LIN {X 0,Y 624.676,Z 1239.512,A -85,B 0,C 180,E1 23145.411,E2 23145.411} C_VEL
LIN {X 0,Y 624.339,Z 1247.75,A -85,B 0,C 180,E1 23143.336,E2 23143.336} C_VEL
LIN {X 0,Y 624.101,Z 1256.133,A -85,B 0,C 180,E1 23140.806,E2 23140.806} C_VEL
LIN {X 0,Y 623.992,Z 1262.422,A -85,B 0,C 180,E1 23138.387,E2 23138.387} C_VEL
LIN {X 0,Y 623.935,Z 1266.954,A -85,B 0,C 180,E1 23136.074,E2 23136.074} C_VEL
LIN {X 0,Y 623.913,Z 1270.232,A -85,B 0,C 180,E1 23133.586,E2 23133.586} C_VEL
LIN {X 0,Y 623.894,Z 1271.702,A -85,B 0,C 180,E1 23131.196,E2 23131.196} C_VEL
LIN {X 0,Y 623.863,Z 1271.839,A -85,B 0,C 180,E1 23129.268,E2 23129.268} C_VEL
LIN {X 0,Y 623.906,Z 1270.982,A -85,B 0,C 180,E1 23127.339,E2 23127.339} C_VEL
LIN {X 0,Y 623.915,Z 1268.958,A -85,B 0,C 180,E1 23125.223,E2 23125.223} C_VEL
LIN {X 0,Y 623.954,Z 1265.168,A -85,B 0,C 180,E1 23122.823,E2 23122.823} C_VEL
LIN {X 0,Y 623.989,Z 1259.714,A -85,B 0,C 180,E1 23120.41,E2 23120.41} C_VEL
LIN {X 0,Y 624.177,Z 1253.512,A -85,B 0,C 180,E1 23118.265,E2 23118.265} C_VEL
LIN {X 0,Y 624.358,Z 1246.696,A -85,B 0,C 180,E1 23116.293,E2 23116.293} C_VEL
LIN {X 0,Y 624.688,Z 1239.108,A -85,B 0,C 180,E1 23114.404,E2 23114.404} C_VEL
LIN {X 0,Y 625.192,Z 1229.451,A -85,B 0,C 180,E1 23112.313,E2 23112.313} C_VEL
LIN {X 0,Y 626.017,Z 1216.16,A -85,B 0,C 180,E1 23109.822,E2 23109.822} C_VEL
LIN {X 0,Y 626.971,Z 1202.854,A -85,B 0,C 180,E1 23107.666,E2 23107.666} C_VEL
LIN {X 0,Y 628.106,Z 1188.914,A -85,B 0,C 180,E1 23105.654,E2 23105.654} C_VEL
LIN {X 0,Y 629.747,Z 1170.474,A -85,B 0,C 180,E1 23103.303,E2 23103.303} C_VEL
LIN {X 0,Y 631.348,Z 1153.818,A -85,B 0,C 180,E1 23101.431,E2 23101.431} C_VEL
LIN {X 0,Y 633.023,Z 1137.229,A -85,B 0,C 180,E1 23099.748,E2 23099.748} C_VEL
LIN {X 0,Y 635.235,Z 1116.148,A -85,B 0,C 180,E1 23097.835,E2 23097.835} C_VEL
LIN {X 0,Y 637.354,Z 1095.911,A -85,B 0,C 180,E1 23096.221,E2 23096.221} C_VEL
LIN {X 0,Y 639.262,Z 1077.648,A -85,B 0,C 180,E1 23094.913,E2 23094.913} C_VEL
LIN {X 0,Y 641.245,Z 1058.295,A -85,B 0,C 180,E1 23093.668,E2 23093.668} C_VEL
LIN {X 0,Y 643.679,Z 1033.574,A -85,B 0,C 180,E1 23092.268,E2 23092.268} C_VEL
LIN {X 0,Y 645.795,Z 1009.706,A -85,B 0,C 180,E1 23091.115,E2 23091.115} C_VEL
LIN {X 0,Y 647.498,Z 989.405,A -85,B 0,C 180,E1 23090.265,E2 23090.265} C_VEL
LIN {X 0,Y 649.072,Z 968.685,A -85,B 0,C 180,E1 23089.516,E2 23089.516} C_VEL
LIN {X 0,Y 650.69,Z 944.811,A -85,B 0,C 180,E1 23088.789,E2 23088.789} C_VEL
LIN {X 0,Y 652.223,Z 916.346,A -85,B 0,C 180,E1 23088.117,E2 23088.117} C_VEL
LIN {X 0,Y 653.175,Z 892.642,A -85,B 0,C 180,E1 23087.705,E2 23087.705} C_VEL
LIN {X 0,Y 657.264,Z 681.046,A -85,B 0,C 180,E1 23084.878,E2 23084.878} C_VEL
LIN {X 0,Y 661.362,Z 477.486,A -85,B 0,C 180,E1 23082.097,E2 23082.097} C_VEL
LIN {X 0,Y 661.477,Z 466.858,A -85,B 0,C 180,E1 23081.939,E2 23081.939} C_VEL
LIN {X 0,Y 648.53,Z 447.721,A -85,B 0,C 180,E1 23080.328,E2 23080.328} C_VEL
LIN {X 0,Y 637.826,Z 432.872,A -85,B 0,C 180,E1 23078.92,E2 23078.92} C_VEL
LIN {X 0,Y 630.127,Z 422.628,A -85,B 0,C 180,E1 23077.858,E2 23077.858} C_VEL
LIN {X 0,Y 627.185,Z 418.313,A -85,B 0,C 180,E1 23077.403,E2 23077.403} C_VEL
LIN {X 0,Y 625.308,Z 415.032,A -85,B 0,C 180,E1 23076.844,E2 23076.844} C_VEL
LIN {X 0,Y 624.947,Z 413.383,A -85,B 0,C 180,E1 23076.607,E2 23076.607} C_VEL
LIN {X 0,Y 624.889,Z 413.367,A -85,B 0,C 180,E1 23073.507,E2 23073.507} C_VEL
LIN {X 0,Y 624.909,Z 413.359,A -85,B 0,C 180,E1 23070.692,E2 23070.692} C_VEL
LIN {X 0,Y 624.895,Z 413.387,A -85,B 0,C 180,E1 23067.441,E2 23067.441} C_VEL
LIN {X 0,Y 624.897,Z 413.361,A -85,B 0,C 180,E1 23064.584,E2 23064.584} C_VEL
LIN {X 0,Y 624.897,Z 413.369,A -85,B 0,C 180,E1 23061.298,E2 23061.298} C_VEL
LIN {X 0,Y 624.89,Z 413.381,A -85,B 0,C 180,E1 23058.471,E2 23058.471} C_VEL
LIN {X 0,Y 624.908,Z 413.351,A -85,B 0,C 180,E1 23055.26,E2 23055.26} C_VEL
LIN {X 0,Y 624.879,Z 413.387,A -85,B 0,C 180,E1 23052.475,E2 23052.475} C_VEL
LIN {X 0,Y 624.948,Z 413.347,A -85,B 0,C 180,E1 23049.392,E2 23049.392} C_VEL
LIN {X 0,Y 624.875,Z 413.388,A -85,B 0,C 180,E1 23046.431,E2 23046.431} C_VEL
LIN {X 0,Y 624.915,Z 413.355,A -85,B 0,C 180,E1 23043.578,E2 23043.578} C_VEL
LIN {X 0,Y 624.883,Z 413.388,A -85,B 0,C 180,E1 23040.458,E2 23040.458} C_VEL
LIN {X 0,Y 624.875,Z 413.369,A -85,B 0,C 180,E1 23037.799,E2 23037.799} C_VEL
LIN {X 0,Y 624.922,Z 413.381,A -85,B 0,C 180,E1 23034.675,E2 23034.675} C_VEL
LIN {X 0,Y 624.866,Z 413.376,A -85,B 0,C 180,E1 23031.905,E2 23031.905} C_VEL
LIN {X 0,Y 624.916,Z 413.371,A -85,B 0,C 180,E1 23029.024,E2 23029.024} C_VEL
LIN {X 0,Y 624.871,Z 413.371,A -85,B 0,C 180,E1 23025.923,E2 23025.923} C_VEL
LIN {X 0,Y 624.871,Z 413.378,A -85,B 0,C 180,E1 23023.26,E2 23023.26} C_VEL
LIN {X 0,Y 624.915,Z 413.353,A -85,B 0,C 180,E1 23020.171,E2 23020.171} C_VEL
LIN {X 0,Y 624.862,Z 413.39,A -85,B 0,C 180,E1 23017.316,E2 23017.316} C_VEL
LIN {X 0,Y 624.923,Z 413.354,A -85,B 0,C 180,E1 23014.405,E2 23014.405} C_VEL
LIN {X 0,Y 624.867,Z 413.387,A -85,B 0,C 180,E1 23011.416,E2 23011.416} C_VEL
LIN {X 0,Y 624.859,Z 413.377,A -85,B 0,C 180,E1 23008.872,E2 23008.872} C_VEL
LIN {X 0,Y 624.933,Z 413.356,A -85,B 0,C 180,E1 23005.833,E2 23005.833} C_VEL
LIN {X 0,Y 624.919,Z 413.433,A -85,B 0,C 180,E1 23004.111,E2 23004.111} C_VEL
LIN {X 0,Y 626.366,Z 417.088,A -85,B 0,C 180,E1 23003.57,E2 23003.57} C_VEL
LIN {X 0,Y 627.307,Z 418.786,A -85,B 0,C 180,E1 23003.29,E2 23003.29} C_VEL
LIN {X 0,Y 631.778,Z 427.462,A -85,B 0,C 180,E1 23001.971,E2 23001.971} C_VEL
LIN {X 0,Y 645.743,Z 446.959,A -85,B 0,C 180,E1 23000.086,E2 23000.086} C_VEL
LIN {X 0,Y 661.259,Z 469.603,A -85,B 0,C 180,E1 22998.147,E2 22998.147} C_VEL
LIN {X 0,Y 661.67,Z 470.762,A -85,B 0,C 180,E1 22998.089,E2 22998.089} C_VEL
LIN {X 0,Y 657.702,Z 668.474,A -85,B 0,C 180,E1 22995.381,E2 22995.381} C_VEL
LIN {X 0,Y 653.463,Z 894.03,A -85,B 0,C 180,E1 22992.376,E2 22992.376} C_VEL
LIN {X 0,Y 652.5,Z 920.141,A -85,B 0,C 180,E1 22991.957,E2 22991.957} C_VEL
LIN {X 0,Y 651.364,Z 942.815,A -85,B 0,C 180,E1 22991.471,E2 22991.471} C_VEL
LIN {X 0,Y 649.955,Z 966.319,A -85,B 0,C 180,E1 22990.835,E2 22990.835} C_VEL
LIN {X 0,Y 647.891,Z 994.546,A -85,B 0,C 180,E1 22989.879,E2 22989.879} C_VEL
LIN {X 0,Y 646.07,Z 1016.552,A -85,B 0,C 180,E1 22988.98,E2 22988.98} C_VEL
LIN {X 0,Y 644.268,Z 1036.777,A -85,B 0,C 180,E1 22988.029,E2 22988.029} C_VEL
LIN {X 0,Y 642.215,Z 1058.311,A -85,B 0,C 180,E1 22986.879,E2 22986.879} C_VEL
LIN {X 0,Y 639.686,Z 1083.572,A -85,B 0,C 180,E1 22985.32,E2 22985.32} C_VEL
LIN {X 0,Y 637.629,Z 1103.286,A -85,B 0,C 180,E1 22983.93,E2 22983.93} C_VEL
LIN {X 0,Y 635.755,Z 1121.099,A -85,B 0,C 180,E1 22982.535,E2 22982.535} C_VEL
LIN {X 0,Y 633.772,Z 1140.151,A -85,B 0,C 180,E1 22980.878,E2 22980.878} C_VEL
LIN {X 0,Y 631.607,Z 1161.096,A -85,B 0,C 180,E1 22978.815,E2 22978.815} C_VEL
LIN {X 0,Y 630.115,Z 1176.719,A -85,B 0,C 180,E1 22977.088,E2 22977.088} C_VEL
LIN {X 0,Y 628.633,Z 1192.732,A -85,B 0,C 180,E1 22975.126,E2 22975.126} C_VEL
LIN {X 0,Y 627.231,Z 1209.562,A -85,B 0,C 180,E1 22972.787,E2 22972.787} C_VEL
LIN {X 0,Y 626.247,Z 1222.456,A -85,B 0,C 180,E1 22970.756,E2 22970.756} C_VEL
LIN {X 0,Y 625.503,Z 1233.839,A -85,B 0,C 180,E1 22968.738,E2 22968.738} C_VEL
LIN {X 0,Y 624.848,Z 1246.152,A -85,B 0,C 180,E1 22966.233,E2 22966.233} C_VEL
LIN {X 0,Y 624.417,Z 1255.1,A -85,B 0,C 180,E1 22964.084,E2 22964.084} C_VEL
LIN {X 0,Y 624.195,Z 1262.149,A -85,B 0,C 180,E1 22962.11,E2 22962.11} C_VEL
LIN {X 0,Y 624.063,Z 1268.064,A -85,B 0,C 180,E1 22960.148,E2 22960.148} C_VEL
LIN {X 0,Y 623.944,Z 1273.567,A -85,B 0,C 180,E1 22957.919,E2 22957.919} C_VEL
LIN {X 0,Y 623.921,Z 1278.057,A -85,B 0,C 180,E1 22955.423,E2 22955.423} C_VEL
LIN {X 0,Y 623.909,Z 1280.61,A -85,B 0,C 180,E1 22953.121,E2 22953.121} C_VEL
LIN {X 0,Y 623.881,Z 1281.738,A -85,B 0,C 180,E1 22951.099,E2 22951.099} C_VEL
LIN {X 0,Y 623.864,Z 1281.826,A -85,B 0,C 180,E1 22949.263,E2 22949.263} C_VEL
LIN {X 0,Y 623.908,Z 1280.945,A -85,B 0,C 180,E1 22947.334,E2 22947.334} C_VEL
LIN {X 0,Y 623.915,Z 1278.896,A -85,B 0,C 180,E1 22945.217,E2 22945.217} C_VEL
LIN {X 0,Y 623.954,Z 1275.074,A -85,B 0,C 180,E1 22942.817,E2 22942.817} C_VEL
LIN {X 0,Y 623.986,Z 1269.831,A -85,B 0,C 180,E1 22940.498,E2 22940.498} C_VEL
LIN {X 0,Y 624.177,Z 1263.348,A -85,B 0,C 180,E1 22938.259,E2 22938.259} C_VEL
LIN {X 0,Y 624.362,Z 1256.506,A -85,B 0,C 180,E1 22936.287,E2 22936.287} C_VEL
LIN {X 0,Y 624.702,Z 1248.892,A -85,B 0,C 180,E1 22934.399,E2 22934.399} C_VEL
LIN {X 0,Y 625.204,Z 1239.21,A -85,B 0,C 180,E1 22932.308,E2 22932.308} C_VEL
LIN {X 0,Y 626.035,Z 1225.866,A -85,B 0,C 180,E1 22929.817,E2 22929.817} C_VEL
LIN {X 0,Y 626.999,Z 1212.519,A -85,B 0,C 180,E1 22927.66,E2 22927.66} C_VEL
LIN {X 0,Y 628.14,Z 1198.554,A -85,B 0,C 180,E1 22925.65,E2 22925.65} C_VEL
LIN {X 0,Y 629.788,Z 1180.051,A -85,B 0,C 180,E1 22923.299,E2 22923.299} C_VEL
LIN {X 0,Y 631.391,Z 1163.362,A -85,B 0,C 180,E1 22921.427,E2 22921.427} C_VEL
LIN {X 0,Y 633.123,Z 1146.25,A -85,B 0,C 180,E1 22919.697,E2 22919.697} C_VEL
LIN {X 0,Y 635.509,Z 1123.455,A -85,B 0,C 180,E1 22917.659,E2 22917.659} C_VEL
LIN {X 0,Y 637.419,Z 1105.273,A -85,B 0,C 180,E1 22916.219,E2 22916.219} C_VEL
LIN {X 0,Y 639.323,Z 1087.025,A -85,B 0,C 180,E1 22914.916,E2 22914.916} C_VEL
LIN {X 0,Y 641.408,Z 1066.727,A -85,B 0,C 180,E1 22913.617,E2 22913.617} C_VEL
LIN {X 0,Y 643.918,Z 1040.682,A -85,B 0,C 180,E1 22912.166,E2 22912.166} C_VEL
LIN {X 0,Y 645.881,Z 1018.687,A -85,B 0,C 180,E1 22911.114,E2 22911.114} C_VEL
LIN {X 0,Y 647.603,Z 998.029,A -85,B 0,C 180,E1 22910.256,E2 22910.256} C_VEL
LIN {X 0,Y 649.276,Z 975.886,A -85,B 0,C 180,E1 22909.466,E2 22909.466} C_VEL
LIN {X 0,Y 651.089,Z 948.263,A -85,B 0,C 180,E1 22908.661,E2 22908.661} C_VEL
LIN {X 0,Y 652.355,Z 923.418,A -85,B 0,C 180,E1 22908.106,E2 22908.106} C_VEL
LIN {X 0,Y 653.235,Z 900.814,A -85,B 0,C 180,E1 22907.723,E2 22907.723} C_VEL
LIN {X 0,Y 657.421,Z 682.788,A -85,B 0,C 180,E1 22904.812,E2 22904.812} C_VEL
LIN {X 0,Y 661.401,Z 483.898,A -85,B 0,C 180,E1 22902.093,E2 22902.093} C_VEL
LIN {X 0,Y 661.549,Z 470.077,A -85,B 0,C 180,E1 22901.888,E2 22901.888} C_VEL
LIN {X 0,Y 647.715,Z 449.878,A -85,B 0,C 180,E1 22900.171,E2 22900.171} C_VEL
LIN {X 0,Y 638.231,Z 436.475,A -85,B 0,C 180,E1 22898.92,E2 22898.92} C_VEL
LIN {X 0,Y 631.264,Z 426.547,A -85,B 0,C 180,E1 22897.921,E2 22897.921} C_VEL
LIN {X 0,Y 627.286,Z 418.676,A -85,B 0,C 180,E1 22896.699,E2 22896.699} C_VEL
LIN {X 0,Y 624.993,Z 413.928,A -85,B 0,C 180,E1 22895.95,E2 22895.95} C_VEL
LIN {X 0,Y 624.895,Z 413.393,A -85,B 0,C 180,E1 22895.848,E2 22895.848} C_VEL
LIN {X 0,Y 624.864,Z 413.376,A -85,B 0,C 180,E1 22893.07,E2 22893.07} C_VEL
LIN {X 0,Y 624.952,Z 413.352,A -85,B 0,C 180,E1 22890.052,E2 22890.052} C_VEL
LIN {X 0,Y 624.877,Z 413.391,A -85,B 0,C 180,E1 22887.132,E2 22887.132} C_VEL
LIN {X 0,Y 624.935,Z 413.364,A -85,B 0,C 180,E1 22884.18,E2 22884.18} C_VEL
LIN {X 0,Y 624.887,Z 413.366,A -85,B 0,C 180,E1 22881.102,E2 22881.102} C_VEL
LIN {X 0,Y 624.916,Z 413.382,A -85,B 0,C 180,E1 22878.277,E2 22878.277} C_VEL
LIN {X 0,Y 624.902,Z 413.351,A -85,B 0,C 180,E1 22875.118,E2 22875.118} C_VEL
LIN {X 0,Y 624.918,Z 413.387,A -85,B 0,C 180,E1 22872.193,E2 22872.193} C_VEL
LIN {X 0,Y 624.91,Z 413.348,A -85,B 0,C 180,E1 22868.929,E2 22868.929} C_VEL
LIN {X 0,Y 624.931,Z 413.389,A -85,B 0,C 180,E1 22865.97,E2 22865.97} C_VEL
LIN {X 0,Y 624.918,Z 413.348,A -85,B 0,C 180,E1 22862.751,E2 22862.751} C_VEL
LIN {X 0,Y 624.957,Z 413.384,A -85,B 0,C 180,E1 22859.633,E2 22859.633} C_VEL
LIN {X 0,Y 624.917,Z 413.35,A -85,B 0,C 180,E1 22856.422,E2 22856.422} C_VEL
LIN {X 0,Y 624.95,Z 413.381,A -85,B 0,C 180,E1 22853.385,E2 22853.385} C_VEL
LIN {X 0,Y 624.923,Z 413.353,A -85,B 0,C 180,E1 22850.235,E2 22850.235} C_VEL
LIN {X 0,Y 624.942,Z 413.378,A -85,B 0,C 180,E1 22847.15,E2 22847.15} C_VEL
LIN {X 0,Y 624.929,Z 413.362,A -85,B 0,C 180,E1 22844.026,E2 22844.026} C_VEL
LIN {X 0,Y 624.936,Z 413.369,A -85,B 0,C 180,E1 22840.95,E2 22840.95} C_VEL
LIN {X 0,Y 624.937,Z 413.377,A -85,B 0,C 180,E1 22837.815,E2 22837.815} C_VEL
LIN {X 0,Y 624.928,Z 413.352,A -85,B 0,C 180,E1 22834.71,E2 22834.71} C_VEL
LIN {X 0,Y 624.944,Z 413.384,A -85,B 0,C 180,E1 22831.628,E2 22831.628} C_VEL
LIN {X 0,Y 624.923,Z 413.373,A -85,B 0,C 180,E1 22828.56,E2 22828.56} C_VEL
LIN {X 0,Y 624.944,Z 413.353,A -85,B 0,C 180,E1 22825.486,E2 22825.486} C_VEL
LIN {X 0,Y 624.983,Z 413.612,A -85,B 0,C 180,E1 22823.248,E2 22823.248} C_VEL
LIN {X 0,Y 626.252,Z 416.878,A -85,B 0,C 180,E1 22822.762,E2 22822.762} C_VEL
LIN {X 0,Y 627.414,Z 418.863,A -85,B 0,C 180,E1 22822.441,E2 22822.441} C_VEL
LIN {X 0,Y 630.527,Z 422.993,A -85,B 0,C 180,E1 22821.998,E2 22821.998} C_VEL
LIN {X 0,Y 643.546,Z 440.758,A -85,B 0,C 180,E1 22820.227,E2 22820.227} C_VEL
LIN {X 0,Y 655.195,Z 457.408,A -85,B 0,C 180,E1 22818.741,E2 22818.741} C_VEL
LIN {X 0,Y 661.581,Z 467.276,A -85,B 0,C 180,E1 22817.954,E2 22817.954} C_VEL
LIN {X 0,Y 660.624,Z 513.045,A -85,B 0,C 180,E1 22817.321,E2 22817.321} C_VEL
LIN {X 0,Y 659.796,Z 520.75,A -85,B 0,C 180,E1 22817.278,E2 22817.278} C_VEL
LIN {X 0,Y 655.117,Z 541.438,A -85,B 0,C 180,E1 22817.395,E2 22817.395} C_VEL
LIN {X 0,Y 654.464,Z 548.048,A -85,B 0,C 180,E1 22817.352,E2 22817.352} C_VEL
LIN {X 0,Y 649.794,Z 770.332,A -85,B 0,C 180,E1 22814.328,E2 22814.328} C_VEL
LIN {X 0,Y 647.174,Z 894.967,A -85,B 0,C 180,E1 22812.648,E2 22812.648} C_VEL
LIN {X 0,Y 645.992,Z 922.208,A -85,B 0,C 180,E1 22812.15,E2 22812.15} C_VEL
LIN {X 0,Y 644.37,Z 948.3,A -85,B 0,C 180,E1 22811.494,E2 22811.494} C_VEL
LIN {X 0,Y 642.811,Z 969.931,A -85,B 0,C 180,E1 22810.822,E2 22810.822} C_VEL
LIN {X 0,Y 641.196,Z 989.829,A -85,B 0,C 180,E1 22810.095,E2 22810.095} C_VEL
LIN {X 0,Y 639.207,Z 1012.325,A -85,B 0,C 180,E1 22809.138,E2 22809.138} C_VEL
LIN {X 0,Y 636.641,Z 1038.744,A -85,B 0,C 180,E1 22807.814,E2 22807.814} C_VEL
LIN {X 0,Y 634.461,Z 1059.319,A -85,B 0,C 180,E1 22806.621,E2 22806.621} C_VEL
LIN {X 0,Y 632.426,Z 1077.897,A -85,B 0,C 180,E1 22805.413,E2 22805.413} C_VEL
LIN {X 0,Y 630.341,Z 1096.659,A -85,B 0,C 180,E1 22804.054,E2 22804.054} C_VEL
LIN {X 0,Y 627.865,Z 1118.735,A -85,B 0,C 180,E1 22802.26,E2 22802.26} C_VEL
LIN {X 0,Y 625.65,Z 1138.333,A -85,B 0,C 180,E1 22800.44,E2 22800.44} C_VEL
LIN {X 0,Y 623.867,Z 1154.814,A -85,B 0,C 180,E1 22798.74,E2 22798.74} C_VEL
LIN {X 0,Y 622,Z 1173.073,A -85,B 0,C 180,E1 22796.646,E2 22796.646} C_VEL
LIN {X 0,Y 620.362,Z 1190.143,A -85,B 0,C 180,E1 22794.403,E2 22794.403} C_VEL
LIN {X 0,Y 619.18,Z 1203.713,A -85,B 0,C 180,E1 22792.404,E2 22792.404} C_VEL
LIN {X 0,Y 618.06,Z 1218.393,A -85,B 0,C 180,E1 22789.959,E2 22789.959} C_VEL
LIN {X 0,Y 617.255,Z 1230.393,A -85,B 0,C 180,E1 22787.635,E2 22787.635} C_VEL
LIN {X 0,Y 616.73,Z 1239.919,A -85,B 0,C 180,E1 22785.518,E2 22785.518} C_VEL
LIN {X 0,Y 616.357,Z 1248.811,A -85,B 0,C 180,E1 22783.225,E2 22783.225} C_VEL
LIN {X 0,Y 616.104,Z 1256.903,A -85,B 0,C 180,E1 22780.664,E2 22780.664} C_VEL
LIN {X 0,Y 615.997,Z 1262.627,A -85,B 0,C 180,E1 22778.403,E2 22778.403} C_VEL
LIN {X 0,Y 615.936,Z 1267.112,A -85,B 0,C 180,E1 22776.059,E2 22776.059} C_VEL
LIN {X 0,Y 615.914,Z 1270.301,A -85,B 0,C 180,E1 22773.539,E2 22773.539} C_VEL
LIN {X 0,Y 615.895,Z 1271.703,A -85,B 0,C 180,E1 22771.212,E2 22771.212} C_VEL
LIN {X 0,Y 615.863,Z 1271.838,A -85,B 0,C 180,E1 22769.259,E2 22769.259} C_VEL
LIN {X 0,Y 615.907,Z 1270.982,A -85,B 0,C 180,E1 22767.304,E2 22767.304} C_VEL
LIN {X 0,Y 615.916,Z 1268.955,A -85,B 0,C 180,E1 22765.16,E2 22765.16} C_VEL
LIN {X 0,Y 615.955,Z 1265.167,A -85,B 0,C 180,E1 22762.729,E2 22762.729} C_VEL
LIN {X 0,Y 616.005,Z 1259.712,A -85,B 0,C 180,E1 22760.284,E2 22760.284} C_VEL
LIN {X 0,Y 616.197,Z 1253.452,A -85,B 0,C 180,E1 22758.092,E2 22758.092} C_VEL
LIN {X 0,Y 616.401,Z 1246.693,A -85,B 0,C 180,E1 22756.112,E2 22756.112} C_VEL
LIN {X 0,Y 616.77,Z 1239.104,A -85,B 0,C 180,E1 22754.199,E2 22754.199} C_VEL
LIN {X 0,Y 617.301,Z 1229.45,A -85,B 0,C 180,E1 22752.08,E2 22752.08} C_VEL
LIN {X 0,Y 618.208,Z 1216.154,A -85,B 0,C 180,E1 22749.556,E2 22749.556} C_VEL
LIN {X 0,Y 619.227,Z 1203.049,A -85,B 0,C 180,E1 22747.403,E2 22747.403} C_VEL
LIN {X 0,Y 620.411,Z 1189.623,A -85,B 0,C 180,E1 22745.434,E2 22745.434} C_VEL
LIN {X 0,Y 622.115,Z 1171.936,A -85,B 0,C 180,E1 22743.129,E2 22743.129} C_VEL
LIN {X 0,Y 623.919,Z 1154.273,A -85,B 0,C 180,E1 22741.111,E2 22741.111} C_VEL
LIN {X 0,Y 625.718,Z 1137.69,A -85,B 0,C 180,E1 22739.406,E2 22739.406} C_VEL
LIN {X 0,Y 628.065,Z 1117.055,A -85,B 0,C 180,E1 22737.505,E2 22737.505} C_VEL
LIN {X 0,Y 630.36,Z 1096.501,A -85,B 0,C 180,E1 22735.844,E2 22735.844} C_VEL
LIN {X 0,Y 632.444,Z 1077.783,A -85,B 0,C 180,E1 22734.489,E2 22734.489} C_VEL
LIN {X 0,Y 634.487,Z 1059.093,A -85,B 0,C 180,E1 22733.275,E2 22733.275} C_VEL
LIN {X 0,Y 636.892,Z 1036.416,A -85,B 0,C 180,E1 22731.966,E2 22731.966} C_VEL
LIN {X 0,Y 639.327,Z 1010.818,A -85,B 0,C 180,E1 22730.704,E2 22730.704} C_VEL
LIN {X 0,Y 641.231,Z 989.385,A -85,B 0,C 180,E1 22729.798,E2 22729.798} C_VEL
LIN {X 0,Y 642.905,Z 968.661,A -85,B 0,C 180,E1 22729.045,E2 22729.045} C_VEL
LIN {X 0,Y 644.623,Z 944.707,A -85,B 0,C 180,E1 22728.313,E2 22728.313} C_VEL
LIN {X 0,Y 646.256,Z 916.125,A -85,B 0,C 180,E1 22727.637,E2 22727.637} C_VEL
LIN {X 0,Y 647.245,Z 892.802,A -85,B 0,C 180,E1 22727.229,E2 22727.229} C_VEL
LIN {X 0,Y 651.579,Z 682.784,A -85,B 0,C 180,E1 22724.401,E2 22724.401} C_VEL
LIN {X 0,Y 655.955,Z 479.443,A -85,B 0,C 180,E1 22721.603,E2 22721.603} C_VEL
LIN {X 0,Y 656.044,Z 470.736,A -85,B 0,C 180,E1 22721.47,E2 22721.47} C_VEL
LIN {X 0,Y 644.58,Z 453.751,A -85,B 0,C 180,E1 22720.015,E2 22720.015} C_VEL
LIN {X 0,Y 633.964,Z 438.914,A -85,B 0,C 180,E1 22718.593,E2 22718.593} C_VEL
LIN {X 0,Y 626.6,Z 429.063,A -85,B 0,C 180,E1 22717.559,E2 22717.559} C_VEL
LIN {X 0,Y 622.58,Z 423.778,A -85,B 0,C 180,E1 22716.975,E2 22716.975} C_VEL
LIN {X 0,Y 619.615,Z 419.636,A -85,B 0,C 180,E1 22716.53,E2 22716.53} C_VEL
LIN {X 0,Y 618.774,Z 418.466,A -85,B 0,C 180,E1 22716.373,E2 22716.373} C_VEL
LIN {X 0,Y 617.079,Z 415.052,A -85,B 0,C 180,E1 22715.8,E2 22715.8} C_VEL
LIN {X 0,Y 616.958,Z 414.367,A -85,B 0,C 180,E1 22715.693,E2 22715.693} C_VEL
LIN {X 0,Y 616.964,Z 414.368,A -85,B 0,C 180,E1 22712.883,E2 22712.883} C_VEL
LIN {X 0,Y 616.964,Z 414.345,A -85,B 0,C 180,E1 22709.624,E2 22709.624} C_VEL
LIN {X 0,Y 616.949,Z 414.367,A -85,B 0,C 180,E1 22706.884,E2 22706.884} C_VEL
LIN {X 0,Y 616.997,Z 414.366,A -85,B 0,C 180,E1 22703.697,E2 22703.697} C_VEL
LIN {X 0,Y 616.939,Z 414.35,A -85,B 0,C 180,E1 22700.889,E2 22700.889} C_VEL
LIN {X 0,Y 617.016,Z 414.374,A -85,B 0,C 180,E1 22697.835,E2 22697.835} C_VEL
LIN {X 0,Y 616.934,Z 414.339,A -85,B 0,C 180,E1 22694.741,E2 22694.741} C_VEL
LIN {X 0,Y 616.989,Z 414.378,A -85,B 0,C 180,E1 22691.834,E2 22691.834} C_VEL
LIN {X 0,Y 616.937,Z 414.34,A -85,B 0,C 180,E1 22688.669,E2 22688.669} C_VEL
LIN {X 0,Y 616.951,Z 414.379,A -85,B 0,C 180,E1 22685.954,E2 22685.954} C_VEL
LIN {X 0,Y 616.951,Z 414.338,A -85,B 0,C 180,E1 22682.694,E2 22682.694} C_VEL
LIN {X 0,Y 616.936,Z 414.379,A -85,B 0,C 180,E1 22680,E2 22680} C_VEL
LIN {X 0,Y 617.001,Z 414.334,A -85,B 0,C 180,E1 22676.934,E2 22676.934} C_VEL
LIN {X 0,Y 616.931,Z 414.38,A -85,B 0,C 180,E1 22673.953,E2 22673.953} C_VEL
LIN {X 0,Y 616.97,Z 414.341,A -85,B 0,C 180,E1 22671.143,E2 22671.143} C_VEL
LIN {X 0,Y 616.939,Z 414.379,A -85,B 0,C 180,E1 22668.027,E2 22668.027} C_VEL
LIN {X 0,Y 616.929,Z 414.347,A -85,B 0,C 180,E1 22665.351,E2 22665.351} C_VEL
LIN {X 0,Y 616.983,Z 414.376,A -85,B 0,C 180,E1 22662.261,E2 22662.261} C_VEL
LIN {X 0,Y 616.92,Z 414.341,A -85,B 0,C 180,E1 22659.408,E2 22659.408} C_VEL
LIN {X 0,Y 616.971,Z 414.378,A -85,B 0,C 180,E1 22656.606,E2 22656.606} C_VEL
LIN {X 0,Y 616.925,Z 414.361,A -85,B 0,C 180,E1 22653.427,E2 22653.427} C_VEL
LIN {X 0,Y 616.928,Z 414.36,A -85,B 0,C 180,E1 22650.801,E2 22650.801} C_VEL
LIN {X 0,Y 616.965,Z 414.379,A -85,B 0,C 180,E1 22647.668,E2 22647.668} C_VEL
LIN {X 0,Y 616.944,Z 414.551,A -85,B 0,C 180,E1 22645.017,E2 22645.017} C_VEL
LIN {X 0,Y 618.251,Z 417.879,A -85,B 0,C 180,E1 22644.507,E2 22644.507} C_VEL
LIN {X 0,Y 619.525,Z 419.947,A -85,B 0,C 180,E1 22644.135,E2 22644.135} C_VEL
LIN {X 0,Y 623.248,Z 427.374,A -85,B 0,C 180,E1 22642.985,E2 22642.985} C_VEL
LIN {X 0,Y 628.893,Z 435.012,A -85,B 0,C 180,E1 22642.17,E2 22642.17} C_VEL
LIN {X 0,Y 639.629,Z 449.917,A -85,B 0,C 180,E1 22640.692,E2 22640.692} C_VEL
LIN {X 0,Y 651.072,Z 466.49,A -85,B 0,C 180,E1 22639.207,E2 22639.207} C_VEL
LIN {X 0,Y 656.233,Z 474.551,A -85,B 0,C 180,E1 22638.558,E2 22638.558} C_VEL
LIN {X 0,Y 652.005,Z 672.031,A -85,B 0,C 180,E1 22635.835,E2 22635.835} C_VEL
LIN {X 0,Y 647.464,Z 896.522,A -85,B 0,C 180,E1 22632.818,E2 22632.818} C_VEL
LIN {X 0,Y 646.505,Z 920.765,A -85,B 0,C 180,E1 22632.422,E2 22632.422} C_VEL
LIN {X 0,Y 645.323,Z 942.96,A -85,B 0,C 180,E1 22631.942,E2 22631.942} C_VEL
LIN {X 0,Y 643.822,Z 966.519,A -85,B 0,C 180,E1 22631.301,E2 22631.301} C_VEL
LIN {X 0,Y 641.694,Z 994.115,A -85,B 0,C 180,E1 22630.362,E2 22630.362} C_VEL
LIN {X 0,Y 639.727,Z 1016.547,A -85,B 0,C 180,E1 22629.441,E2 22629.441} C_VEL
LIN {X 0,Y 637.81,Z 1036.774,A -85,B 0,C 180,E1 22628.484,E2 22628.484} C_VEL
LIN {X 0,Y 635.625,Z 1058.312,A -85,B 0,C 180,E1 22627.326,E2 22627.326} C_VEL
LIN {X 0,Y 632.919,Z 1083.442,A -85,B 0,C 180,E1 22625.764,E2 22625.764} C_VEL
LIN {X 0,Y 630.705,Z 1103.283,A -85,B 0,C 180,E1 22624.355,E2 22624.355} C_VEL
LIN {X 0,Y 628.711,Z 1121.097,A -85,B 0,C 180,E1 22622.945,E2 22622.945} C_VEL
LIN {X 0,Y 626.544,Z 1140.527,A -85,B 0,C 180,E1 22621.238,E2 22621.238} C_VEL
LIN {X 0,Y 624.259,Z 1161.001,A -85,B 0,C 180,E1 22619.197,E2 22619.197} C_VEL
LIN {X 0,Y 622.638,Z 1176.717,A -85,B 0,C 180,E1 22617.44,E2 22617.44} C_VEL
LIN {X 0,Y 621.022,Z 1193.073,A -85,B 0,C 180,E1 22615.411,E2 22615.411} C_VEL
LIN {X 0,Y 619.473,Z 1210.209,A -85,B 0,C 180,E1 22612.988,E2 22612.988} C_VEL
LIN {X 0,Y 618.417,Z 1223.027,A -85,B 0,C 180,E1 22610.932,E2 22610.932} C_VEL
LIN {X 0,Y 617.588,Z 1234.866,A -85,B 0,C 180,E1 22608.791,E2 22608.791} C_VEL
LIN {X 0,Y 616.896,Z 1246.863,A -85,B 0,C 180,E1 22606.281,E2 22606.281} C_VEL
LIN {X 0,Y 616.459,Z 1255.458,A -85,B 0,C 180,E1 22604.174,E2 22604.174} C_VEL
LIN {X 0,Y 616.215,Z 1262.456,A -85,B 0,C 180,E1 22602.174,E2 22602.174} C_VEL
LIN {X 0,Y 616.074,Z 1268.32,A -85,B 0,C 180,E1 22600.186,E2 22600.186} C_VEL
LIN {X 0,Y 615.948,Z 1273.766,A -85,B 0,C 180,E1 22597.928,E2 22597.928} C_VEL
LIN {X 0,Y 615.922,Z 1278.182,A -85,B 0,C 180,E1 22595.4,E2 22595.4} C_VEL
LIN {X 0,Y 615.91,Z 1280.678,A -85,B 0,C 180,E1 22593.068,E2 22593.068} C_VEL
LIN {X 0,Y 615.882,Z 1281.737,A -85,B 0,C 180,E1 22591.114,E2 22591.114} C_VEL
LIN {X 0,Y 615.864,Z 1281.826,A -85,B 0,C 180,E1 22589.253,E2 22589.253} C_VEL
LIN {X 0,Y 615.909,Z 1280.945,A -85,B 0,C 180,E1 22587.299,E2 22587.299} C_VEL
LIN {X 0,Y 615.915,Z 1279.006,A -85,B 0,C 180,E1 22585.248,E2 22585.248} C_VEL
LIN {X 0,Y 615.956,Z 1275.246,A -85,B 0,C 180,E1 22582.817,E2 22582.817} C_VEL
LIN {X 0,Y 616.003,Z 1269.831,A -85,B 0,C 180,E1 22580.373,E2 22580.373} C_VEL
LIN {X 0,Y 616.198,Z 1263.305,A -85,B 0,C 180,E1 22578.092,E2 22578.092} C_VEL
LIN {X 0,Y 616.407,Z 1256.505,A -85,B 0,C 180,E1 22576.107,E2 22576.107} C_VEL
LIN {X 0,Y 616.785,Z 1248.893,A -85,B 0,C 180,E1 22574.194,E2 22574.194} C_VEL
LIN {X 0,Y 617.315,Z 1239.212,A -85,B 0,C 180,E1 22572.074,E2 22572.074} C_VEL
LIN {X 0,Y 618.227,Z 1225.864,A -85,B 0,C 180,E1 22569.551,E2 22569.551} C_VEL
LIN {X 0,Y 619.257,Z 1212.729,A -85,B 0,C 180,E1 22567.399,E2 22567.399} C_VEL
LIN {X 0,Y 620.508,Z 1198.556,A -85,B 0,C 180,E1 22565.331,E2 22565.331} C_VEL
LIN {X 0,Y 622.309,Z 1180.049,A -85,B 0,C 180,E1 22562.952,E2 22562.952} C_VEL
LIN {X 0,Y 624.012,Z 1163.36,A -85,B 0,C 180,E1 22561.057,E2 22561.057} C_VEL
LIN {X 0,Y 625.882,Z 1146.226,A -85,B 0,C 180,E1 22559.307,E2 22559.307} C_VEL
LIN {X 0,Y 628.452,Z 1123.456,A -85,B 0,C 180,E1 22557.25,E2 22557.25} C_VEL
LIN {X 0,Y 630.498,Z 1105.204,A -85,B 0,C 180,E1 22555.791,E2 22555.791} C_VEL
LIN {X 0,Y 632.486,Z 1087.352,A -85,B 0,C 180,E1 22554.505,E2 22554.505} C_VEL
LIN {X 0,Y 634.568,Z 1068.346,A -85,B 0,C 180,E1 22553.274,E2 22553.274} C_VEL
LIN {X 0,Y 637.072,Z 1044.66,A -85,B 0,C 180,E1 22551.915,E2 22551.915} C_VEL
LIN {X 0,Y 639.417,Z 1019.813,A -85,B 0,C 180,E1 22550.704,E2 22550.704} C_VEL
LIN {X 0,Y 641.28,Z 998.794,A -85,B 0,C 180,E1 22549.82,E2 22549.82} C_VEL
LIN {X 0,Y 643.004,Z 977.363,A -85,B 0,C 180,E1 22549.046,E2 22549.046} C_VEL
LIN {X 0,Y 644.878,Z 951.16,A -85,B 0,C 180,E1 22548.259,E2 22548.259} C_VEL
LIN {X 0,Y 646.338,Z 924.367,A -85,B 0,C 180,E1 22547.648,E2 22547.648} C_VEL
LIN {X 0,Y 647.278,Z 901.852,A -85,B 0,C 180,E1 22547.26,E2 22547.26} C_VEL
LIN {X 0,Y 651.677,Z 687.876,A -85,B 0,C 180,E1 22544.38,E2 22544.38} C_VEL
LIN {X 0,Y 655.942,Z 487.874,A -85,B 0,C 180,E1 22541.628,E2 22541.628} C_VEL
LIN {X 0,Y 656.171,Z 474.102,A -85,B 0,C 180,E1 22541.429,E2 22541.429} C_VEL
LIN {X 0,Y 643.564,Z 455.604,A -85,B 0,C 180,E1 22539.83,E2 22539.83} C_VEL
LIN {X 0,Y 634.499,Z 442.691,A -85,B 0,C 180,E1 22538.612,E2 22538.612} C_VEL
LIN {X 0,Y 626.861,Z 432.216,A -85,B 0,C 180,E1 22537.54,E2 22537.54} C_VEL
LIN {X 0,Y 622.613,Z 426.43,A -85,B 0,C 180,E1 22536.892,E2 22536.892} C_VEL
LIN {X 0,Y 620.63,Z 422.358,A -85,B 0,C 180,E1 22536.247,E2 22536.247} C_VEL
LIN {X 0,Y 618.731,Z 418.514,A -85,B 0,C 180,E1 22535.623,E2 22535.623} C_VEL
LIN {X 0,Y 617.109,Z 415.346,A -85,B 0,C 180,E1 22535.09,E2 22535.09} C_VEL
LIN {X 0,Y 616.929,Z 414.358,A -85,B 0,C 180,E1 22534.95,E2 22534.95} C_VEL
LIN {X 0,Y 616.969,Z 414.378,A -85,B 0,C 180,E1 22531.784,E2 22531.784} C_VEL
LIN {X 0,Y 616.933,Z 414.359,A -85,B 0,C 180,E1 22528.987,E2 22528.987} C_VEL
LIN {X 0,Y 617.008,Z 414.34,A -85,B 0,C 180,E1 22525.948,E2 22525.948} C_VEL
LIN {X 0,Y 616.943,Z 414.38,A -85,B 0,C 180,E1 22522.991,E2 22522.991} C_VEL
LIN {X 0,Y 616.998,Z 414.339,A -85,B 0,C 180,E1 22520.094,E2 22520.094} C_VEL
LIN {X 0,Y 616.955,Z 414.376,A -85,B 0,C 180,E1 22516.961,E2 22516.961} C_VEL
LIN {X 0,Y 617.005,Z 414.34,A -85,B 0,C 180,E1 22513.973,E2 22513.973} C_VEL
LIN {X 0,Y 616.965,Z 414.37,A -85,B 0,C 180,E1 22510.836,E2 22510.836} C_VEL
LIN {X 0,Y 617.008,Z 414.345,A -85,B 0,C 180,E1 22507.824,E2 22507.824} C_VEL
LIN {X 0,Y 616.971,Z 414.365,A -85,B 0,C 180,E1 22504.648,E2 22504.648} C_VEL
LIN {X 0,Y 617.01,Z 414.35,A -85,B 0,C 180,E1 22501.579,E2 22501.579} C_VEL
LIN {X 0,Y 616.98,Z 414.363,A -85,B 0,C 180,E1 22498.514,E2 22498.514} C_VEL
LIN {X 0,Y 617.008,Z 414.354,A -85,B 0,C 180,E1 22495.352,E2 22495.352} C_VEL
LIN {X 0,Y 616.985,Z 414.357,A -85,B 0,C 180,E1 22492.27,E2 22492.27} C_VEL
LIN {X 0,Y 617.004,Z 414.361,A -85,B 0,C 180,E1 22489.129,E2 22489.129} C_VEL
LIN {X 0,Y 616.988,Z 414.349,A -85,B 0,C 180,E1 22486.027,E2 22486.027} C_VEL
LIN {X 0,Y 617,Z 414.373,A -85,B 0,C 180,E1 22482.943,E2 22482.943} C_VEL
LIN {X 0,Y 616.994,Z 414.34,A -85,B 0,C 180,E1 22479.771,E2 22479.771} C_VEL
LIN {X 0,Y 616.995,Z 414.373,A -85,B 0,C 180,E1 22476.708,E2 22476.708} C_VEL
LIN {X 0,Y 617.002,Z 414.347,A -85,B 0,C 180,E1 22473.535,E2 22473.535} C_VEL
LIN {X 0,Y 616.988,Z 414.346,A -85,B 0,C 180,E1 22470.484,E2 22470.484} C_VEL
LIN {X 0,Y 617.012,Z 414.371,A -85,B 0,C 180,E1 22467.341,E2 22467.341} C_VEL
LIN {X 0,Y 616.99,Z 414.397,A -85,B 0,C 180,E1 22464.187,E2 22464.187} C_VEL
LIN {X 0,Y 618.4,Z 417.978,A -85,B 0,C 180,E1 22463.632,E2 22463.632} C_VEL
LIN {X 0,Y 619.599,Z 419.577,A -85,B 0,C 180,E1 22463.381,E2 22463.381} C_VEL
LIN {X 0,Y 622.694,Z 423.85,A -85,B 0,C 180,E1 22462.918,E2 22462.918} C_VEL
LIN {X 0,Y 624.623,Z 426.485,A -85,B 0,C 180,E1 22462.634,E2 22462.634} C_VEL
LIN {X 0,Y 631.753,Z 435.847,A -85,B 0,C 180,E1 22461.623,E2 22461.623} C_VEL
LIN {X 0,Y 642.236,Z 450.414,A -85,B 0,C 180,E1 22460.202,E2 22460.202} C_VEL
LIN {X 0,Y 653.575,Z 466.942,A -85,B 0,C 180,E1 22458.747,E2 22458.747} C_VEL
LIN {X 0,Y 656.146,Z 471.183,A -85,B 0,C 180,E1 22458.422,E2 22458.422} C_VEL
LIN {X 0,Y 654.464,Z 548.048,A -85,B 0,C 180,E1 22457.352,E2 22457.352} C_VEL
LIN {X 0,Y 653.62,Z 555.753,A -85,B 0,C 180,E1 22457.31,E2 22457.31} C_VEL
LIN {X 0,Y 648.904,Z 576.427,A -85,B 0,C 180,E1 22457.432,E2 22457.432} C_VEL
LIN {X 0,Y 648.23,Z 583.037,A -85,B 0,C 180,E1 22457.391,E2 22457.391} C_VEL
LIN {X 0,Y 643.477,Z 798.613,A -85,B 0,C 180,E1 22454.445,E2 22454.445} C_VEL
LIN {X 0,Y 641.285,Z 895.125,A -85,B 0,C 180,E1 22453.132,E2 22453.132} C_VEL
LIN {X 0,Y 640.028,Z 922.455,A -85,B 0,C 180,E1 22452.629,E2 22452.629} C_VEL
LIN {X 0,Y 638.323,Z 948.397,A -85,B 0,C 180,E1 22451.973,E2 22451.973} C_VEL
LIN {X 0,Y 636.683,Z 969.946,A -85,B 0,C 180,E1 22451.3,E2 22451.3} C_VEL
LIN {X 0,Y 634.971,Z 989.842,A -85,B 0,C 180,E1 22450.569,E2 22450.569} C_VEL
LIN {X 0,Y 632.964,Z 1011.205,A -85,B 0,C 180,E1 22449.658,E2 22449.658} C_VEL
LIN {X 0,Y 630.265,Z 1037.604,A -85,B 0,C 180,E1 22448.34,E2 22448.34} C_VEL
LIN {X 0,Y 627.815,Z 1059.402,A -85,B 0,C 180,E1 22447.068,E2 22447.068} C_VEL
LIN {X 0,Y 625.664,Z 1077.83,A -85,B 0,C 180,E1 22445.86,E2 22445.86} C_VEL
LIN {X 0,Y 623.419,Z 1096.815,A -85,B 0,C 180,E1 22444.472,E2 22444.472} C_VEL
LIN {X 0,Y 620.779,Z 1118.913,A -85,B 0,C 180,E1 22442.657,E2 22442.657} C_VEL
LIN {X 0,Y 618.417,Z 1138.339,A -85,B 0,C 180,E1 22440.835,E2 22440.835} C_VEL
LIN {X 0,Y 616.551,Z 1154.356,A -85,B 0,C 180,E1 22439.167,E2 22439.167} C_VEL
LIN {X 0,Y 614.657,Z 1171.818,A -85,B 0,C 180,E1 22437.148,E2 22437.148} C_VEL
LIN {X 0,Y 612.846,Z 1189.026,A -85,B 0,C 180,E1 22434.886,E2 22434.886} C_VEL
LIN {X 0,Y 611.573,Z 1202.446,A -85,B 0,C 180,E1 22432.901,E2 22432.901} C_VEL
LIN {X 0,Y 610.444,Z 1215.605,A -85,B 0,C 180,E1 22430.722,E2 22430.722} C_VEL
LIN {X 0,Y 609.45,Z 1229.001,A -85,B 0,C 180,E1 22428.165,E2 22428.165} C_VEL
LIN {X 0,Y 608.887,Z 1238.706,A -85,B 0,C 180,E1 22426.017,E2 22426.017} C_VEL
LIN {X 0,Y 608.452,Z 1246.693,A -85,B 0,C 180,E1 22423.981,E2 22423.981} C_VEL
LIN {X 0,Y 608.214,Z 1253.509,A -85,B 0,C 180,E1 22421.957,E2 22421.957} C_VEL
LIN {X 0,Y 608.005,Z 1260.219,A -85,B 0,C 180,E1 22419.563,E2 22419.563} C_VEL
LIN {X 0,Y 607.951,Z 1265.673,A -85,B 0,C 180,E1 22416.993,E2 22416.993} C_VEL
LIN {X 0,Y 607.914,Z 1269.063,A -85,B 0,C 180,E1 22414.72,E2 22414.72} C_VEL
LIN {X 0,Y 607.908,Z 1271.048,A -85,B 0,C 180,E1 22412.548,E2 22412.548} C_VEL
LIN {X 0,Y 607.877,Z 1271.905,A -85,B 0,C 180,E1 22410.38,E2 22410.38} C_VEL
LIN {X 0,Y 607.907,Z 1271.319,A -85,B 0,C 180,E1 22407.74,E2 22407.74} C_VEL
LIN {X 0,Y 607.914,Z 1269.289,A -85,B 0,C 180,E1 22405.378,E2 22405.378} C_VEL
LIN {X 0,Y 607.941,Z 1265.994,A -85,B 0,C 180,E1 22403.107,E2 22403.107} C_VEL
LIN {X 0,Y 607.987,Z 1260.927,A -85,B 0,C 180,E1 22400.633,E2 22400.633} C_VEL
LIN {X 0,Y 608.212,Z 1253.81,A -85,B 0,C 180,E1 22398.048,E2 22398.048} C_VEL
LIN {X 0,Y 608.436,Z 1247.043,A -85,B 0,C 180,E1 22396.024,E2 22396.024} C_VEL
LIN {X 0,Y 608.859,Z 1239.101,A -85,B 0,C 180,E1 22393.988,E2 22393.988} C_VEL
LIN {X 0,Y 609.434,Z 1229.251,A -85,B 0,C 180,E1 22391.798,E2 22391.798} C_VEL
LIN {X 0,Y 610.406,Z 1216.148,A -85,B 0,C 180,E1 22389.283,E2 22389.283} C_VEL
LIN {X 0,Y 611.515,Z 1203.042,A -85,B 0,C 180,E1 22387.102,E2 22387.102} C_VEL
LIN {X 0,Y 612.787,Z 1189.618,A -85,B 0,C 180,E1 22385.108,E2 22385.108} C_VEL
LIN {X 0,Y 614.622,Z 1172.149,A -85,B 0,C 180,E1 22382.802,E2 22382.802} C_VEL
LIN {X 0,Y 616.542,Z 1154.443,A -85,B 0,C 180,E1 22380.753,E2 22380.753} C_VEL
LIN {X 0,Y 618.43,Z 1138.228,A -85,B 0,C 180,E1 22379.064,E2 22379.064} C_VEL
LIN {X 0,Y 620.949,Z 1117.65,A -85,B 0,C 180,E1 22377.14,E2 22377.14} C_VEL
LIN {X 0,Y 623.458,Z 1096.49,A -85,B 0,C 180,E1 22375.413,E2 22375.413} C_VEL
LIN {X 0,Y 625.685,Z 1077.697,A -85,B 0,C 180,E1 22374.04,E2 22374.04} C_VEL
LIN {X 0,Y 627.956,Z 1058.163,A -85,B 0,C 180,E1 22372.764,E2 22372.764} C_VEL
LIN {X 0,Y 630.697,Z 1033.555,A -85,B 0,C 180,E1 22371.35,E2 22371.35} C_VEL
LIN {X 0,Y 633.109,Z 1009.669,A -85,B 0,C 180,E1 22370.183,E2 22370.183} C_VEL
LIN {X 0,Y 635.014,Z 989.366,A -85,B 0,C 180,E1 22369.322,E2 22369.322} C_VEL
LIN {X 0,Y 636.783,Z 968.639,A -85,B 0,C 180,E1 22368.565,E2 22368.565} C_VEL
LIN {X 0,Y 638.572,Z 944.994,A -85,B 0,C 180,E1 22367.839,E2 22367.839} C_VEL
LIN {X 0,Y 640.311,Z 916.392,A -85,B 0,C 180,E1 22367.158,E2 22367.158} C_VEL
LIN {X 0,Y 641.355,Z 893.099,A -85,B 0,C 180,E1 22366.747,E2 22366.747} C_VEL
LIN {X 0,Y 645.962,Z 683.853,A -85,B 0,C 180,E1 22363.907,E2 22363.907} C_VEL
LIN {X 0,Y 650.624,Z 480.37,A -85,B 0,C 180,E1 22361.086,E2 22361.086} C_VEL
LIN {X 0,Y 650.657,Z 474.688,A -85,B 0,C 180,E1 22360.995,E2 22360.995} C_VEL
LIN {X 0,Y 640.651,Z 459.768,A -85,B 0,C 180,E1 22359.698,E2 22359.698} C_VEL
LIN {X 0,Y 630.125,Z 444.94,A -85,B 0,C 180,E1 22358.262,E2 22358.262} C_VEL
LIN {X 0,Y 623.105,Z 435.503,A -85,B 0,C 180,E1 22357.259,E2 22357.259} C_VEL
LIN {X 0,Y 618.701,Z 429.769,A -85,B 0,C 180,E1 22356.609,E2 22356.609} C_VEL
LIN {X 0,Y 615.182,Z 424.965,A -85,B 0,C 180,E1 22356.071,E2 22356.071} C_VEL
LIN {X 0,Y 612.017,Z 420.793,A -85,B 0,C 180,E1 22355.579,E2 22355.579} C_VEL
LIN {X 0,Y 610.082,Z 418.461,A -85,B 0,C 180,E1 22355.234,E2 22355.234} C_VEL
LIN {X 0,Y 609.044,Z 415.33,A -85,B 0,C 180,E1 22354.728,E2 22354.728} C_VEL
LIN {X 0,Y 609.019,Z 415.355,A -85,B 0,C 180,E1 22351.569,E2 22351.569} C_VEL
LIN {X 0,Y 609.023,Z 415.351,A -85,B 0,C 180,E1 22348.754,E2 22348.754} C_VEL
LIN {X 0,Y 609.02,Z 415.327,A -85,B 0,C 180,E1 22345.458,E2 22345.458} C_VEL
LIN {X 0,Y 609.016,Z 415.371,A -85,B 0,C 180,E1 22342.593,E2 22342.593} C_VEL
LIN {X 0,Y 609.023,Z 415.34,A -85,B 0,C 180,E1 22339.269,E2 22339.269} C_VEL
LIN {X 0,Y 609.007,Z 415.359,A -85,B 0,C 180,E1 22336.501,E2 22336.501} C_VEL
LIN {X 0,Y 609.057,Z 415.339,A -85,B 0,C 180,E1 22333.384,E2 22333.384} C_VEL
LIN {X 0,Y 608.998,Z 415.353,A -85,B 0,C 180,E1 22330.405,E2 22330.405} C_VEL
LIN {X 0,Y 609.07,Z 415.342,A -85,B 0,C 180,E1 22327.262,E2 22327.262} C_VEL
LIN {X 0,Y 608.994,Z 415.351,A -85,B 0,C 180,E1 22324.237,E2 22324.237} C_VEL
LIN {X 0,Y 609.074,Z 415.342,A -85,B 0,C 180,E1 22321.129,E2 22321.129} C_VEL
LIN {X 0,Y 608.993,Z 415.352,A -85,B 0,C 180,E1 22318.118,E2 22318.118} C_VEL
LIN {X 0,Y 609.057,Z 415.342,A -85,B 0,C 180,E1 22315.103,E2 22315.103} C_VEL
LIN {X 0,Y 608.994,Z 415.353,A -85,B 0,C 180,E1 22312.073,E2 22312.073} C_VEL
LIN {X 0,Y 609.007,Z 415.346,A -85,B 0,C 180,E1 22309.308,E2 22309.308} C_VEL
LIN {X 0,Y 609.001,Z 415.345,A -85,B 0,C 180,E1 22306.034,E2 22306.034} C_VEL
LIN {X 0,Y 608.992,Z 415.355,A -85,B 0,C 180,E1 22303.302,E2 22303.302} C_VEL
LIN {X 0,Y 609.031,Z 415.327,A -85,B 0,C 180,E1 22300.132,E2 22300.132} C_VEL
LIN {X 0,Y 608.986,Z 415.368,A -85,B 0,C 180,E1 22297.304,E2 22297.304} C_VEL
LIN {X 0,Y 609.053,Z 415.327,A -85,B 0,C 180,E1 22294.316,E2 22294.316} C_VEL
LIN {X 0,Y 608.986,Z 415.362,A -85,B 0,C 180,E1 22291.351,E2 22291.351} C_VEL
LIN {X 0,Y 608.987,Z 415.353,A -85,B 0,C 180,E1 22288.746,E2 22288.746} C_VEL
LIN {X 0,Y 609.069,Z 415.438,A -85,B 0,C 180,E1 22285.98,E2 22285.98} C_VEL
LIN {X 0,Y 610.263,Z 418.749,A -85,B 0,C 180,E1 22285.465,E2 22285.465} C_VEL
LIN {X 0,Y 611.494,Z 420.769,A -85,B 0,C 180,E1 22285.089,E2 22285.089} C_VEL
LIN {X 0,Y 613.561,Z 424.593,A -85,B 0,C 180,E1 22284.424,E2 22284.424} C_VEL
LIN {X 0,Y 614.779,Z 427.223,A -85,B 0,C 180,E1 22284.046,E2 22284.046} C_VEL
LIN {X 0,Y 625.436,Z 441.527,A -85,B 0,C 180,E1 22282.459,E2 22282.459} C_VEL
LIN {X 0,Y 635.953,Z 456.224,A -85,B 0,C 180,E1 22280.987,E2 22280.987} C_VEL
LIN {X 0,Y 647.494,Z 473.116,A -85,B 0,C 180,E1 22279.463,E2 22279.463} C_VEL
LIN {X 0,Y 650.837,Z 478.47,A -85,B 0,C 180,E1 22279.033,E2 22279.033} C_VEL
LIN {X 0,Y 646.343,Z 675.637,A -85,B 0,C 180,E1 22276.296,E2 22276.296} C_VEL
LIN {X 0,Y 641.538,Z 898.035,A -85,B 0,C 180,E1 22273.283,E2 22273.283} C_VEL
LIN {X 0,Y 640.565,Z 921.138,A -85,B 0,C 180,E1 22272.9,E2 22272.9} C_VEL
LIN {X 0,Y 639.328,Z 943.098,A -85,B 0,C 180,E1 22272.422,E2 22272.422} C_VEL
LIN {X 0,Y 637.725,Z 966.878,A -85,B 0,C 180,E1 22271.771,E2 22271.771} C_VEL
LIN {X 0,Y 635.434,Z 994.842,A -85,B 0,C 180,E1 22270.81,E2 22270.81} C_VEL
LIN {X 0,Y 633.392,Z 1016.9,A -85,B 0,C 180,E1 22269.895,E2 22269.895} C_VEL
LIN {X 0,Y 631.397,Z 1036.77,A -85,B 0,C 180,E1 22268.948,E2 22268.948} C_VEL
LIN {X 0,Y 629.167,Z 1057.483,A -85,B 0,C 180,E1 22267.828,E2 22267.828} C_VEL
LIN {X 0,Y 626.283,Z 1082.597,A -85,B 0,C 180,E1 22266.268,E2 22266.268} C_VEL
LIN {X 0,Y 623.816,Z 1103.281,A -85,B 0,C 180,E1 22264.788,E2 22264.788} C_VEL
LIN {X 0,Y 621.691,Z 1121.095,A -85,B 0,C 180,E1 22263.366,E2 22263.366} C_VEL
LIN {X 0,Y 619.382,Z 1140.527,A -85,B 0,C 180,E1 22261.64,E2 22261.64} C_VEL
LIN {X 0,Y 616.941,Z 1160.99,A -85,B 0,C 180,E1 22259.579,E2 22259.579} C_VEL
LIN {X 0,Y 615.176,Z 1176.715,A -85,B 0,C 180,E1 22257.802,E2 22257.802} C_VEL
LIN {X 0,Y 613.494,Z 1192.728,A -85,B 0,C 180,E1 22255.791,E2 22255.791} C_VEL
LIN {X 0,Y 611.774,Z 1210.211,A -85,B 0,C 180,E1 22253.295,E2 22253.295} C_VEL
LIN {X 0,Y 610.638,Z 1223.025,A -85,B 0,C 180,E1 22251.212,E2 22251.212} C_VEL
LIN {X 0,Y 609.755,Z 1234.865,A -85,B 0,C 180,E1 22249.042,E2 22249.042} C_VEL
LIN {X 0,Y 608.959,Z 1247.275,A -85,B 0,C 180,E1 22246.401,E2 22246.401} C_VEL
LIN {X 0,Y 608.502,Z 1255.817,A -85,B 0,C 180,E1 22244.266,E2 22244.266} C_VEL
LIN {X 0,Y 608.235,Z 1262.76,A -85,B 0,C 180,E1 22242.24,E2 22242.24} C_VEL
LIN {X 0,Y 608.084,Z 1268.573,A -85,B 0,C 180,E1 22240.226,E2 22240.226} C_VEL
LIN {X 0,Y 607.946,Z 1274.157,A -85,B 0,C 180,E1 22237.843,E2 22237.843} C_VEL
LIN {X 0,Y 607.922,Z 1278.432,A -85,B 0,C 180,E1 22235.282,E2 22235.282} C_VEL
LIN {X 0,Y 607.911,Z 1280.746,A -85,B 0,C 180,E1 22233.014,E2 22233.014} C_VEL
LIN {X 0,Y 607.876,Z 1281.76,A -85,B 0,C 180,E1 22231.034,E2 22231.034} C_VEL
LIN {X 0,Y 607.867,Z 1281.804,A -85,B 0,C 180,E1 22229.149,E2 22229.149} C_VEL
LIN {X 0,Y 607.91,Z 1280.945,A -85,B 0,C 180,E1 22227.263,E2 22227.263} C_VEL
LIN {X 0,Y 607.917,Z 1279.003,A -85,B 0,C 180,E1 22225.186,E2 22225.186} C_VEL
LIN {X 0,Y 607.958,Z 1275.418,A -85,B 0,C 180,E1 22222.817,E2 22222.817} C_VEL
LIN {X 0,Y 608.012,Z 1270.084,A -85,B 0,C 180,E1 22220.341,E2 22220.341} C_VEL
LIN {X 0,Y 608.216,Z 1263.533,A -85,B 0,C 180,E1 22218.006,E2 22218.006} C_VEL
LIN {X 0,Y 608.443,Z 1256.857,A -85,B 0,C 180,E1 22216.018,E2 22216.018} C_VEL
LIN {X 0,Y 608.874,Z 1248.892,A -85,B 0,C 180,E1 22213.983,E2 22213.983} C_VEL
LIN {X 0,Y 609.448,Z 1239.021,A -85,B 0,C 180,E1 22211.794,E2 22211.794} C_VEL
LIN {X 0,Y 610.427,Z 1225.862,A -85,B 0,C 180,E1 22209.278,E2 22209.278} C_VEL
LIN {X 0,Y 611.546,Z 1212.727,A -85,B 0,C 180,E1 22207.098,E2 22207.098} C_VEL
LIN {X 0,Y 612.822,Z 1199.268,A -85,B 0,C 180,E1 22205.103,E2 22205.103} C_VEL
LIN {X 0,Y 614.666,Z 1181.737,A -85,B 0,C 180,E1 22202.798,E2 22202.798} C_VEL
LIN {X 0,Y 616.559,Z 1164.284,A -85,B 0,C 180,E1 22200.78,E2 22200.78} C_VEL
LIN {X 0,Y 618.456,Z 1148.005,A -85,B 0,C 180,E1 22199.087,E2 22199.087} C_VEL
LIN {X 0,Y 620.923,Z 1127.855,A -85,B 0,C 180,E1 22197.203,E2 22197.203} C_VEL
LIN {X 0,Y 623.45,Z 1106.536,A -85,B 0,C 180,E1 22195.461,E2 22195.461} C_VEL
LIN {X 0,Y 625.674,Z 1087.754,A -85,B 0,C 180,E1 22194.09,E2 22194.09} C_VEL
LIN {X 0,Y 627.935,Z 1068.343,A -85,B 0,C 180,E1 22192.821,E2 22192.821} C_VEL
LIN {X 0,Y 630.674,Z 1043.832,A -85,B 0,C 180,E1 22191.409,E2 22191.409} C_VEL
LIN {X 0,Y 633.096,Z 1019.81,A -85,B 0,C 180,E1 22190.234,E2 22190.234} C_VEL
LIN {X 0,Y 635.055,Z 998.898,A -85,B 0,C 180,E1 22189.349,E2 22189.349} C_VEL
LIN {X 0,Y 636.828,Z 978.099,A -85,B 0,C 180,E1 22188.592,E2 22188.592} C_VEL
LIN {X 0,Y 638.714,Z 953.183,A -85,B 0,C 180,E1 22187.832,E2 22187.832} C_VEL
LIN {X 0,Y 640.356,Z 925.479,A -85,B 0,C 180,E1 22187.185,E2 22187.185} C_VEL
LIN {X 0,Y 641.37,Z 902.676,A -85,B 0,C 180,E1 22186.786,E2 22186.786} C_VEL
LIN {X 0,Y 645.915,Z 695.292,A -85,B 0,C 180,E1 22183.973,E2 22183.973} C_VEL
LIN {X 0,Y 650.52,Z 492.148,A -85,B 0,C 180,E1 22181.16,E2 22181.16} C_VEL
LIN {X 0,Y 650.721,Z 477.958,A -85,B 0,C 180,E1 22180.947,E2 22180.947} C_VEL
LIN {X 0,Y 637.056,Z 457.744,A -85,B 0,C 180,E1 22179.162,E2 22179.162} C_VEL
LIN {X 0,Y 623.481,Z 438.788,A -85,B 0,C 180,E1 22177.258,E2 22177.258} C_VEL
LIN {X 0,Y 614.237,Z 426.27,A -85,B 0,C 180,E1 22175.838,E2 22175.838} C_VEL
LIN {X 0,Y 612.848,Z 423.68,A -85,B 0,C 180,E1 22175.394,E2 22175.394} C_VEL
LIN {X 0,Y 610.925,Z 419.621,A -85,B 0,C 180,E1 22174.72,E2 22174.72} C_VEL
LIN {X 0,Y 609.247,Z 416.326,A -85,B 0,C 180,E1 22174.145,E2 22174.145} C_VEL
LIN {X 0,Y 609.042,Z 415.331,A -85,B 0,C 180,E1 22173.995,E2 22173.995} C_VEL
LIN {X 0,Y 608.991,Z 415.35,A -85,B 0,C 180,E1 22171.034,E2 22171.034} C_VEL
LIN {X 0,Y 609.073,Z 415.361,A -85,B 0,C 180,E1 22167.967,E2 22167.967} C_VEL
LIN {X 0,Y 608.998,Z 415.333,A -85,B 0,C 180,E1 22164.958,E2 22164.958} C_VEL
LIN {X 0,Y 609.081,Z 415.348,A -85,B 0,C 180,E1 22161.879,E2 22161.879} C_VEL
LIN {X 0,Y 609.01,Z 415.357,A -85,B 0,C 180,E1 22158.772,E2 22158.772} C_VEL
LIN {X 0,Y 609.078,Z 415.326,A -85,B 0,C 180,E1 22155.716,E2 22155.716} C_VEL
LIN {X 0,Y 609.021,Z 415.363,A -85,B 0,C 180,E1 22152.613,E2 22152.613} C_VEL
LIN {X 0,Y 609.072,Z 415.319,A -85,B 0,C 180,E1 22149.449,E2 22149.449} C_VEL
LIN {X 0,Y 609.031,Z 415.365,A -85,B 0,C 180,E1 22146.315,E2 22146.315} C_VEL
LIN {X 0,Y 609.063,Z 415.318,A -85,B 0,C 180,E1 22143.106,E2 22143.106} C_VEL
LIN {X 0,Y 609.047,Z 415.366,A -85,B 0,C 180,E1 22140,E2 22140} C_VEL
LIN {X 0,Y 609.055,Z 415.319,A -85,B 0,C 180,E1 22136.706,E2 22136.706} C_VEL
LIN {X 0,Y 609.075,Z 415.361,A -85,B 0,C 180,E1 22133.496,E2 22133.496} C_VEL
LIN {X 0,Y 609.046,Z 415.325,A -85,B 0,C 180,E1 22130.265,E2 22130.265} C_VEL
LIN {X 0,Y 609.064,Z 415.354,A -85,B 0,C 180,E1 22127.099,E2 22127.099} C_VEL
LIN {X 0,Y 609.051,Z 415.336,A -85,B 0,C 180,E1 22123.99,E2 22123.99} C_VEL
LIN {X 0,Y 609.059,Z 415.345,A -85,B 0,C 180,E1 22120.931,E2 22120.931} C_VEL
LIN {X 0,Y 609.062,Z 415.355,A -85,B 0,C 180,E1 22117.714,E2 22117.714} C_VEL
LIN {X 0,Y 609.052,Z 415.325,A -85,B 0,C 180,E1 22114.548,E2 22114.548} C_VEL
LIN {X 0,Y 609.07,Z 415.35,A -85,B 0,C 180,E1 22111.356,E2 22111.356} C_VEL
LIN {X 0,Y 609.056,Z 415.357,A -85,B 0,C 180,E1 22108.198,E2 22108.198} C_VEL
LIN {X 0,Y 609.086,Z 415.468,A -85,B 0,C 180,E1 22105.131,E2 22105.131} C_VEL
LIN {X 0,Y 610.486,Z 419.029,A -85,B 0,C 180,E1 22104.563,E2 22104.563} C_VEL
LIN {X 0,Y 612.797,Z 422.065,A -85,B 0,C 180,E1 22104.2,E2 22104.2} C_VEL
LIN {X 0,Y 616.587,Z 426.803,A -85,B 0,C 180,E1 22103.621,E2 22103.621} C_VEL
LIN {X 0,Y 628.204,Z 442.245,A -85,B 0,C 180,E1 22101.919,E2 22101.919} C_VEL
LIN {X 0,Y 638.675,Z 456.943,A -85,B 0,C 180,E1 22100.476,E2 22100.476} C_VEL
LIN {X 0,Y 649.507,Z 472.828,A -85,B 0,C 180,E1 22099.062,E2 22099.062} C_VEL
LIN {X 0,Y 650.75,Z 475.225,A -85,B 0,C 180,E1 22098.896,E2 22098.896} C_VEL
LIN {X 0,Y 648.23,Z 583.037,A -85,B 0,C 180,E1 22097.391,E2 22097.391} C_VEL
LIN {X 0,Y 647.369,Z 590.741,A -85,B 0,C 180,E1 22097.35,E2 22097.35} C_VEL
LIN {X 0,Y 642.657,Z 611.41,A -85,B 0,C 180,E1 22097.474,E2 22097.474} C_VEL
LIN {X 0,Y 641.977,Z 618.019,A -85,B 0,C 180,E1 22097.433,E2 22097.433} C_VEL
LIN {X 0,Y 636.941,Z 835.952,A -85,B 0,C 180,E1 22094.445,E2 22094.445} C_VEL
LIN {X 0,Y 635.39,Z 896.806,A -85,B 0,C 180,E1 22093.602,E2 22093.602} C_VEL
LIN {X 0,Y 633.902,Z 925.605,A -85,B 0,C 180,E1 22093.048,E2 22093.048} C_VEL
LIN {X 0,Y 632.271,Z 949.162,A -85,B 0,C 180,E1 22092.441,E2 22092.441} C_VEL
LIN {X 0,Y 630.601,Z 969.962,A -85,B 0,C 180,E1 22091.787,E2 22091.787} C_VEL
LIN {X 0,Y 628.797,Z 989.855,A -85,B 0,C 180,E1 22091.053,E2 22091.053} C_VEL
LIN {X 0,Y 626.68,Z 1011.216,A -85,B 0,C 180,E1 22090.136,E2 22090.136} C_VEL
LIN {X 0,Y 623.808,Z 1037.613,A -85,B 0,C 180,E1 22088.81,E2 22088.81} C_VEL
LIN {X 0,Y 621.223,Z 1059.334,A -85,B 0,C 180,E1 22087.534,E2 22087.534} C_VEL
LIN {X 0,Y 618.836,Z 1078.645,A -85,B 0,C 180,E1 22086.255,E2 22086.255} C_VEL
LIN {X 0,Y 616.253,Z 1099.336,A -85,B 0,C 180,E1 22084.717,E2 22084.717} C_VEL
LIN {X 0,Y 613.278,Z 1122.248,A -85,B 0,C 180,E1 22082.773,E2 22082.773} C_VEL
LIN {X 0,Y 611.094,Z 1139.357,A -85,B 0,C 180,E1 22081.136,E2 22081.136} C_VEL
LIN {X 0,Y 609.061,Z 1155.748,A -85,B 0,C 180,E1 22079.399,E2 22079.399} C_VEL
LIN {X 0,Y 606.857,Z 1174.621,A -85,B 0,C 180,E1 22077.157,E2 22077.157} C_VEL
LIN {X 0,Y 605.103,Z 1190.369,A -85,B 0,C 180,E1 22075.027,E2 22075.027} C_VEL
LIN {X 0,Y 603.757,Z 1203.718,A -85,B 0,C 180,E1 22073.009,E2 22073.009} C_VEL
LIN {X 0,Y 602.443,Z 1218.39,A -85,B 0,C 180,E1 22070.502,E2 22070.502} C_VEL
LIN {X 0,Y 601.49,Z 1230.401,A -85,B 0,C 180,E1 22068.113,E2 22068.113} C_VEL
LIN {X 0,Y 600.899,Z 1239.921,A -85,B 0,C 180,E1 22065.938,E2 22065.938} C_VEL
LIN {X 0,Y 600.423,Z 1248.813,A -85,B 0,C 180,E1 22063.582,E2 22063.582} C_VEL
LIN {X 0,Y 600.135,Z 1256.908,A -85,B 0,C 180,E1 22060.951,E2 22060.951} C_VEL
LIN {X 0,Y 600.005,Z 1262.623,A -85,B 0,C 180,E1 22058.628,E2 22058.628} C_VEL
LIN {X 0,Y 599.942,Z 1267.108,A -85,B 0,C 180,E1 22056.222,E2 22056.222} C_VEL
LIN {X 0,Y 599.913,Z 1270.301,A -85,B 0,C 180,E1 22053.634,E2 22053.634} C_VEL
LIN {X 0,Y 599.898,Z 1271.703,A -85,B 0,C 180,E1 22051.244,E2 22051.244} C_VEL
LIN {X 0,Y 599.864,Z 1271.838,A -85,B 0,C 180,E1 22049.239,E2 22049.239} C_VEL
LIN {X 0,Y 599.908,Z 1270.981,A -85,B 0,C 180,E1 22047.232,E2 22047.232} C_VEL
LIN {X 0,Y 599.918,Z 1269.061,A -85,B 0,C 180,E1 22045.127,E2 22045.127} C_VEL
LIN {X 0,Y 599.958,Z 1265.508,A -85,B 0,C 180,E1 22042.726,E2 22042.726} C_VEL
LIN {X 0,Y 600.023,Z 1260.217,A -85,B 0,C 180,E1 22040.217,E2 22040.217} C_VEL
LIN {X 0,Y 600.244,Z 1253.505,A -85,B 0,C 180,E1 22037.79,E2 22037.79} C_VEL
LIN {X 0,Y 600.518,Z 1246.591,A -85,B 0,C 180,E1 22035.711,E2 22035.711} C_VEL
LIN {X 0,Y 600.975,Z 1238.692,A -85,B 0,C 180,E1 22033.673,E2 22033.673} C_VEL
LIN {X 0,Y 601.62,Z 1228.515,A -85,B 0,C 180,E1 22031.395,E2 22031.395} C_VEL
LIN {X 0,Y 602.702,Z 1215.029,A -85,B 0,C 180,E1 22028.807,E2 22028.807} C_VEL
LIN {X 0,Y 603.881,Z 1202.401,A -85,B 0,C 180,E1 22026.693,E2 22026.693} C_VEL
LIN {X 0,Y 605.277,Z 1188.674,A -85,B 0,C 180,E1 22024.639,E2 22024.639} C_VEL
LIN {X 0,Y 607.345,Z 1170.451,A -85,B 0,C 180,E1 22022.235,E2 22022.235} C_VEL
LIN {X 0,Y 609.206,Z 1154.48,A -85,B 0,C 180,E1 22020.371,E2 22020.371} C_VEL
LIN {X 0,Y 611.177,Z 1138.727,A -85,B 0,C 180,E1 22018.711,E2 22018.711} C_VEL
LIN {X 0,Y 613.684,Z 1119.39,A -85,B 0,C 180,E1 22016.875,E2 22016.875} C_VEL
LIN {X 0,Y 616.517,Z 1097.08,A -85,B 0,C 180,E1 22015.018,E2 22015.018} C_VEL
LIN {X 0,Y 618.868,Z 1078.42,A -85,B 0,C 180,E1 22013.639,E2 22013.639} C_VEL
LIN {X 0,Y 621.254,Z 1059.085,A -85,B 0,C 180,E1 22012.36,E2 22012.36} C_VEL
LIN {X 0,Y 624.07,Z 1035.485,A -85,B 0,C 180,E1 22010.98,E2 22010.98} C_VEL
LIN {X 0,Y 626.722,Z 1010.782,A -85,B 0,C 180,E1 22009.754,E2 22009.754} C_VEL
LIN {X 0,Y 628.847,Z 989.346,A -85,B 0,C 180,E1 22008.837,E2 22008.837} C_VEL
LIN {X 0,Y 630.647,Z 969.358,A -85,B 0,C 180,E1 22008.101,E2 22008.101} C_VEL
LIN {X 0,Y 632.416,Z 947.234,A -85,B 0,C 180,E1 22007.413,E2 22007.413} C_VEL
LIN {X 0,Y 634.27,Z 919.517,A -85,B 0,C 180,E1 22006.725,E2 22006.725} C_VEL
LIN {X 0,Y 635.481,Z 894.225,A -85,B 0,C 180,E1 22006.269,E2 22006.269} C_VEL
LIN {X 0,Y 639.114,Z 740.026,A -85,B 0,C 180,E1 22004.16,E2 22004.16} C_VEL
LIN {X 0,Y 644.226,Z 526.541,A -85,B 0,C 180,E1 22001.2,E2 22001.2} C_VEL
LIN {X 0,Y 645.327,Z 478.519,A -85,B 0,C 180,E1 22000.512,E2 22000.512} C_VEL
LIN {X 0,Y 633.42,Z 460.929,A -85,B 0,C 180,E1 21998.923,E2 21998.923} C_VEL
LIN {X 0,Y 620.006,Z 442.369,A -85,B 0,C 180,E1 21997.01,E2 21997.01} C_VEL
LIN {X 0,Y 611.623,Z 431.303,A -85,B 0,C 180,E1 21995.735,E2 21995.735} C_VEL
LIN {X 0,Y 603.728,Z 421.282,A -85,B 0,C 180,E1 21994.472,E2 21994.472} C_VEL
LIN {X 0,Y 601.929,Z 418.942,A -85,B 0,C 180,E1 21994.157,E2 21994.157} C_VEL
LIN {X 0,Y 601.085,Z 416.322,A -85,B 0,C 180,E1 21993.731,E2 21993.731} C_VEL
LIN {X 0,Y 601.079,Z 416.324,A -85,B 0,C 180,E1 21990.877,E2 21990.877} C_VEL
LIN {X 0,Y 601.087,Z 416.355,A -85,B 0,C 180,E1 21987.545,E2 21987.545} C_VEL
LIN {X 0,Y 601.075,Z 416.321,A -85,B 0,C 180,E1 21984.679,E2 21984.679} C_VEL
LIN {X 0,Y 601.086,Z 416.33,A -85,B 0,C 180,E1 21981.365,E2 21981.365} C_VEL
LIN {X 0,Y 601.071,Z 416.347,A -85,B 0,C 180,E1 21978.526,E2 21978.526} C_VEL
LIN {X 0,Y 601.099,Z 416.312,A -85,B 0,C 180,E1 21975.337,E2 21975.337} C_VEL
LIN {X 0,Y 601.064,Z 416.354,A -85,B 0,C 180,E1 21972.473,E2 21972.473} C_VEL
LIN {X 0,Y 601.128,Z 416.307,A -85,B 0,C 180,E1 21969.382,E2 21969.382} C_VEL
LIN {X 0,Y 601.06,Z 416.356,A -85,B 0,C 180,E1 21966.399,E2 21966.399} C_VEL
LIN {X 0,Y 601.123,Z 416.308,A -85,B 0,C 180,E1 21963.338,E2 21963.338} C_VEL
LIN {X 0,Y 601.06,Z 416.356,A -85,B 0,C 180,E1 21960.286,E2 21960.286} C_VEL
LIN {X 0,Y 601.087,Z 416.317,A -85,B 0,C 180,E1 21957.426,E2 21957.426} C_VEL
LIN {X 0,Y 601.06,Z 416.357,A -85,B 0,C 180,E1 21954.176,E2 21954.176} C_VEL
LIN {X 0,Y 601.061,Z 416.323,A -85,B 0,C 180,E1 21951.486,E2 21951.486} C_VEL
LIN {X 0,Y 601.074,Z 416.357,A -85,B 0,C 180,E1 21948.193,E2 21948.193} C_VEL
LIN {X 0,Y 601.047,Z 416.322,A -85,B 0,C 180,E1 21945.451,E2 21945.451} C_VEL
LIN {X 0,Y 601.119,Z 416.353,A -85,B 0,C 180,E1 21942.368,E2 21942.368} C_VEL
LIN {X 0,Y 601.043,Z 416.315,A -85,B 0,C 180,E1 21939.348,E2 21939.348} C_VEL
LIN {X 0,Y 601.123,Z 416.344,A -85,B 0,C 180,E1 21936.367,E2 21936.367} C_VEL
LIN {X 0,Y 601.043,Z 416.338,A -85,B 0,C 180,E1 21933.285,E2 21933.285} C_VEL
LIN {X 0,Y 601.08,Z 416.324,A -85,B 0,C 180,E1 21930.449,E2 21930.449} C_VEL
LIN {X 0,Y 601.05,Z 416.35,A -85,B 0,C 180,E1 21927.271,E2 21927.271} C_VEL
LIN {X 0,Y 601.072,Z 416.575,A -85,B 0,C 180,E1 21926.983,E2 21926.983} C_VEL
LIN {X 0,Y 602.439,Z 419.914,A -85,B 0,C 180,E1 21926.418,E2 21926.418} C_VEL
LIN {X 0,Y 603.633,Z 421.604,A -85,B 0,C 180,E1 21926.067,E2 21926.067} C_VEL
LIN {X 0,Y 605.552,Z 425.474,A -85,B 0,C 180,E1 21925.388,E2 21925.388} C_VEL
LIN {X 0,Y 606.498,Z 427.352,A -85,B 0,C 180,E1 21925.134,E2 21925.134} C_VEL
LIN {X 0,Y 614.074,Z 437.283,A -85,B 0,C 180,E1 21923.94,E2 21923.94} C_VEL
LIN {X 0,Y 622.382,Z 448.588,A -85,B 0,C 180,E1 21922.694,E2 21922.694} C_VEL
LIN {X 0,Y 632.288,Z 462.523,A -85,B 0,C 180,E1 21921.285,E2 21921.285} C_VEL
LIN {X 0,Y 643.952,Z 479.761,A -85,B 0,C 180,E1 21919.72,E2 21919.72} C_VEL
LIN {X 0,Y 645.487,Z 482.321,A -85,B 0,C 180,E1 21919.517,E2 21919.517} C_VEL
LIN {X 0,Y 640.714,Z 679.703,A -85,B 0,C 180,E1 21916.759,E2 21916.759} C_VEL
LIN {X 0,Y 635.654,Z 899.609,A -85,B 0,C 180,E1 21913.755,E2 21913.755} C_VEL
LIN {X 0,Y 634.662,Z 921.668,A -85,B 0,C 180,E1 21913.384,E2 21913.384} C_VEL
LIN {X 0,Y 633.383,Z 943.229,A -85,B 0,C 180,E1 21912.911,E2 21912.911} C_VEL
LIN {X 0,Y 631.704,Z 966.833,A -85,B 0,C 180,E1 21912.262,E2 21912.262} C_VEL
LIN {X 0,Y 629.315,Z 994.539,A -85,B 0,C 180,E1 21911.307,E2 21911.307} C_VEL
LIN {X 0,Y 627.176,Z 1016.542,A -85,B 0,C 180,E1 21910.391,E2 21910.391} C_VEL
LIN {X 0,Y 625.14,Z 1035.762,A -85,B 0,C 180,E1 21909.473,E2 21909.473} C_VEL
LIN {X 0,Y 622.957,Z 1054.948,A -85,B 0,C 180,E1 21908.438,E2 21908.438} C_VEL
LIN {X 0,Y 620.578,Z 1074.849,A -85,B 0,C 180,E1 21907.23,E2 21907.23} C_VEL
LIN {X 0,Y 617.508,Z 1099.273,A -85,B 0,C 180,E1 21905.537,E2 21905.537} C_VEL
LIN {X 0,Y 614.968,Z 1118.907,A -85,B 0,C 180,E1 21903.981,E2 21903.981} C_VEL
LIN {X 0,Y 612.777,Z 1136.092,A -85,B 0,C 180,E1 21902.464,E2 21902.464} C_VEL
LIN {X 0,Y 610.545,Z 1154.042,A -85,B 0,C 180,E1 21900.706,E2 21900.706} C_VEL
LIN {X 0,Y 608.061,Z 1174.177,A -85,B 0,C 180,E1 21898.477,E2 21898.477} C_VEL
LIN {X 0,Y 606.249,Z 1189.644,A -85,B 0,C 180,E1 21896.544,E2 21896.544} C_VEL
LIN {X 0,Y 604.634,Z 1204.913,A -85,B 0,C 180,E1 21894.416,E2 21894.416} C_VEL
LIN {X 0,Y 603.094,Z 1220.72,A -85,B 0,C 180,E1 21891.899,E2 21891.899} C_VEL
LIN {X 0,Y 602.125,Z 1232.289,A -85,B 0,C 180,E1 21889.798,E2 21889.798} C_VEL
LIN {X 0,Y 601.342,Z 1242.924,A -85,B 0,C 180,E1 21887.611,E2 21887.611} C_VEL
LIN {X 0,Y 600.694,Z 1254.031,A -85,B 0,C 180,E1 21884.948,E2 21884.948} C_VEL
LIN {X 0,Y 600.3,Z 1262.151,A -85,B 0,C 180,E1 21882.6,E2 21882.6} C_VEL
LIN {X 0,Y 600.114,Z 1268.065,A -85,B 0,C 180,E1 21880.557,E2 21880.557} C_VEL
LIN {X 0,Y 599.99,Z 1273.351,A -85,B 0,C 180,E1 21878.333,E2 21878.333} C_VEL
LIN {X 0,Y 599.935,Z 1277.787,A -85,B 0,C 180,E1 21875.832,E2 21875.832} C_VEL
LIN {X 0,Y 599.91,Z 1280.542,A -85,B 0,C 180,E1 21873.341,E2 21873.341} C_VEL
LIN {X 0,Y 599.891,Z 1281.715,A -85,B 0,C 180,E1 21871.239,E2 21871.239} C_VEL
LIN {X 0,Y 599.864,Z 1281.826,A -85,B 0,C 180,E1 21869.233,E2 21869.233} C_VEL
LIN {X 0,Y 599.908,Z 1281.013,A -85,B 0,C 180,E1 21867.322,E2 21867.322} C_VEL
LIN {X 0,Y 599.917,Z 1279.114,A -85,B 0,C 180,E1 21865.217,E2 21865.217} C_VEL
LIN {X 0,Y 599.959,Z 1275.586,A -85,B 0,C 180,E1 21862.817,E2 21862.817} C_VEL
LIN {X 0,Y 600.031,Z 1270.084,A -85,B 0,C 180,E1 21860.211,E2 21860.211} C_VEL
LIN {X 0,Y 600.238,Z 1263.65,A -85,B 0,C 180,E1 21857.882,E2 21857.882} C_VEL
LIN {X 0,Y 600.501,Z 1256.856,A -85,B 0,C 180,E1 21855.83,E2 21855.83} C_VEL
LIN {X 0,Y 600.97,Z 1248.793,A -85,B 0,C 180,E1 21853.743,E2 21853.743} C_VEL
LIN {X 0,Y 601.604,Z 1238.749,A -85,B 0,C 180,E1 21851.489,E2 21851.489} C_VEL
LIN {X 0,Y 602.683,Z 1225.287,A -85,B 0,C 180,E1 21848.897,E2 21848.897} C_VEL
LIN {X 0,Y 603.858,Z 1212.666,A -85,B 0,C 180,E1 21846.78,E2 21846.78} C_VEL
LIN {X 0,Y 605.292,Z 1198.56,A -85,B 0,C 180,E1 21844.667,E2 21844.667} C_VEL
LIN {X 0,Y 607.39,Z 1180.045,A -85,B 0,C 180,E1 21842.231,E2 21842.231} C_VEL
LIN {X 0,Y 609.266,Z 1163.976,A -85,B 0,C 180,E1 21840.36,E2 21840.36} C_VEL
LIN {X 0,Y 611.308,Z 1147.747,A -85,B 0,C 180,E1 21838.657,E2 21838.657} C_VEL
LIN {X 0,Y 613.996,Z 1127.086,A -85,B 0,C 180,E1 21836.714,E2 21836.714} C_VEL
LIN {X 0,Y 616.655,Z 1105.866,A -85,B 0,C 180,E1 21834.969,E2 21834.969} C_VEL
LIN {X 0,Y 619.034,Z 1087.016,A -85,B 0,C 180,E1 21833.586,E2 21833.586} C_VEL
LIN {X 0,Y 621.637,Z 1065.906,A -85,B 0,C 180,E1 21832.204,E2 21832.204} C_VEL
LIN {X 0,Y 624.593,Z 1040.675,A -85,B 0,C 180,E1 21830.776,E2 21830.776} C_VEL
LIN {X 0,Y 626.825,Z 1019.806,A -85,B 0,C 180,E1 21829.755,E2 21829.755} C_VEL
LIN {X 0,Y 628.827,Z 999.529,A -85,B 0,C 180,E1 21828.889,E2 21828.889} C_VEL
LIN {X 0,Y 630.693,Z 978.836,A -85,B 0,C 180,E1 21828.129,E2 21828.129} C_VEL
LIN {X 0,Y 632.514,Z 955.986,A -85,B 0,C 180,E1 21827.421,E2 21827.421} C_VEL
LIN {X 0,Y 634.38,Z 927.338,A -85,B 0,C 180,E1 21826.728,E2 21826.728} C_VEL
LIN {X 0,Y 635.5,Z 903.715,A -85,B 0,C 180,E1 21826.306,E2 21826.306} C_VEL
LIN {X 0,Y 640.219,Z 701.25,A -85,B 0,C 180,E1 21823.538,E2 21823.538} C_VEL
LIN {X 0,Y 645.164,Z 495.481,A -85,B 0,C 180,E1 21820.67,E2 21820.67} C_VEL
LIN {X 0,Y 645.378,Z 481.85,A -85,B 0,C 180,E1 21820.464,E2 21820.464} C_VEL
LIN {X 0,Y 629.832,Z 458.814,A -85,B 0,C 180,E1 21818.37,E2 21818.37} C_VEL
LIN {X 0,Y 616.29,Z 440.142,A -85,B 0,C 180,E1 21816.399,E2 21816.399} C_VEL
LIN {X 0,Y 608.631,Z 430.203,A -85,B 0,C 180,E1 21815.215,E2 21815.215} C_VEL
LIN {X 0,Y 605.839,Z 425.969,A -85,B 0,C 180,E1 21814.708,E2 21814.708} C_VEL
LIN {X 0,Y 603.626,Z 421.561,A -85,B 0,C 180,E1 21813.934,E2 21813.934} C_VEL
LIN {X 0,Y 601.3,Z 417.567,A -85,B 0,C 180,E1 21813.168,E2 21813.168} C_VEL
LIN {X 0,Y 601.053,Z 416.338,A -85,B 0,C 180,E1 21812.956,E2 21812.956} C_VEL
LIN {X 0,Y 601.102,Z 416.317,A -85,B 0,C 180,E1 21809.826,E2 21809.826} C_VEL
LIN {X 0,Y 601.061,Z 416.347,A -85,B 0,C 180,E1 21806.903,E2 21806.903} C_VEL
LIN {X 0,Y 601.12,Z 416.338,A -85,B 0,C 180,E1 21803.737,E2 21803.737} C_VEL
LIN {X 0,Y 601.066,Z 416.322,A -85,B 0,C 180,E1 21800.787,E2 21800.787} C_VEL
LIN {X 0,Y 601.133,Z 416.352,A -85,B 0,C 180,E1 21797.618,E2 21797.618} C_VEL
LIN {X 0,Y 601.074,Z 416.313,A -85,B 0,C 180,E1 21794.548,E2 21794.548} C_VEL
LIN {X 0,Y 601.131,Z 416.346,A -85,B 0,C 180,E1 21791.416,E2 21791.416} C_VEL
LIN {X 0,Y 601.088,Z 416.315,A -85,B 0,C 180,E1 21788.321,E2 21788.321} C_VEL
LIN {X 0,Y 601.13,Z 416.342,A -85,B 0,C 180,E1 21785.153,E2 21785.153} C_VEL
LIN {X 0,Y 601.105,Z 416.319,A -85,B 0,C 180,E1 21782.002,E2 21782.002} C_VEL
LIN {X 0,Y 601.11,Z 416.341,A -85,B 0,C 180,E1 21778.666,E2 21778.666} C_VEL
LIN {X 0,Y 601.129,Z 416.324,A -85,B 0,C 180,E1 21775.516,E2 21775.516} C_VEL
LIN {X 0,Y 601.11,Z 416.332,A -85,B 0,C 180,E1 21772.353,E2 21772.353} C_VEL
LIN {X 0,Y 601.126,Z 416.334,A -85,B 0,C 180,E1 21769.166,E2 21769.166} C_VEL
LIN {X 0,Y 601.111,Z 416.322,A -85,B 0,C 180,E1 21766.043,E2 21766.043} C_VEL
LIN {X 0,Y 601.123,Z 416.35,A -85,B 0,C 180,E1 21762.877,E2 21762.877} C_VEL
LIN {X 0,Y 601.118,Z 416.312,A -85,B 0,C 180,E1 21759.656,E2 21759.656} C_VEL
LIN {X 0,Y 601.124,Z 416.349,A -85,B 0,C 180,E1 21756.471,E2 21756.471} C_VEL
LIN {X 0,Y 601.131,Z 416.328,A -85,B 0,C 180,E1 21753.207,E2 21753.207} C_VEL
LIN {X 0,Y 601.138,Z 416.312,A -85,B 0,C 180,E1 21749.956,E2 21749.956} C_VEL
LIN {X 0,Y 601.107,Z 416.331,A -85,B 0,C 180,E1 21746.706,E2 21746.706} C_VEL
LIN {X 0,Y 601.136,Z 416.491,A -85,B 0,C 180,E1 21746.136,E2 21746.136} C_VEL
LIN {X 0,Y 602.423,Z 419.779,A -85,B 0,C 180,E1 21745.644,E2 21745.644} C_VEL
LIN {X 0,Y 605.064,Z 422.897,A -85,B 0,C 180,E1 21745.215,E2 21745.215} C_VEL
LIN {X 0,Y 609.777,Z 429.019,A -85,B 0,C 180,E1 21744.458,E2 21744.458} C_VEL
LIN {X 0,Y 613.535,Z 433.801,A -85,B 0,C 180,E1 21743.875,E2 21743.875} C_VEL
LIN {X 0,Y 624.672,Z 448.64,A -85,B 0,C 180,E1 21742.218,E2 21742.218} C_VEL
LIN {X 0,Y 635.405,Z 463.877,A -85,B 0,C 180,E1 21740.714,E2 21740.714} C_VEL
LIN {X 0,Y 645.414,Z 478.639,A -85,B 0,C 180,E1 21739.387,E2 21739.387} C_VEL
LIN {X 0,Y 641.977,Z 618.019,A -85,B 0,C 180,E1 21737.433,E2 21737.433} C_VEL
LIN {X 0,Y 641.103,Z 625.725,A -85,B 0,C 180,E1 21737.393,E2 21737.393} C_VEL
LIN {X 0,Y 636.375,Z 646.392,A -85,B 0,C 180,E1 21737.52,E2 21737.52} C_VEL
LIN {X 0,Y 635.701,Z 653.001,A -85,B 0,C 180,E1 21737.478,E2 21737.478} C_VEL
LIN {X 0,Y 630.296,Z 876.839,A -85,B 0,C 180,E1 21734.4,E2 21734.4} C_VEL
LIN {X 0,Y 629.056,Z 907.954,A -85,B 0,C 180,E1 21733.914,E2 21733.914} C_VEL
LIN {X 0,Y 627.71,Z 930.183,A -85,B 0,C 180,E1 21733.441,E2 21733.441} C_VEL
LIN {X 0,Y 626.143,Z 951.444,A -85,B 0,C 180,E1 21732.874,E2 21732.874} C_VEL
LIN {X 0,Y 624.374,Z 972.197,A -85,B 0,C 180,E1 21732.207,E2 21732.207} C_VEL
LIN {X 0,Y 622.188,Z 995.004,A -85,B 0,C 180,E1 21731.339,E2 21731.339} C_VEL
LIN {X 0,Y 619.387,Z 1020.881,A -85,B 0,C 180,E1 21730.161,E2 21730.161} C_VEL
LIN {X 0,Y 616.856,Z 1042.029,A -85,B 0,C 180,E1 21729.038,E2 21729.038} C_VEL
LIN {X 0,Y 614.429,Z 1061.255,A -85,B 0,C 180,E1 21727.883,E2 21727.883} C_VEL
LIN {X 0,Y 611.866,Z 1080.854,A -85,B 0,C 180,E1 21726.56,E2 21726.56} C_VEL
LIN {X 0,Y 608.711,Z 1104.457,A -85,B 0,C 180,E1 21724.751,E2 21724.751} C_VEL
LIN {X 0,Y 606.026,Z 1123.846,A -85,B 0,C 180,E1 21723.054,E2 21723.054} C_VEL
LIN {X 0,Y 603.791,Z 1140.376,A -85,B 0,C 180,E1 21721.444,E2 21721.444} C_VEL
LIN {X 0,Y 601.527,Z 1157.604,A -85,B 0,C 180,E1 21719.585,E2 21719.585} C_VEL
LIN {X 0,Y 599.09,Z 1176.963,A -85,B 0,C 180,E1 21717.215,E2 21717.215} C_VEL
LIN {X 0,Y 597.43,Z 1191.072,A -85,B 0,C 180,E1 21715.265,E2 21715.265} C_VEL
LIN {X 0,Y 595.943,Z 1204.99,A -85,B 0,C 180,E1 21713.119,E2 21713.119} C_VEL
LIN {X 0,Y 594.507,Z 1219.972,A -85,B 0,C 180,E1 21710.477,E2 21710.477} C_VEL
LIN {X 0,Y 593.589,Z 1230.861,A -85,B 0,C 180,E1 21708.261,E2 21708.261} C_VEL
LIN {X 0,Y 592.99,Z 1239.923,A -85,B 0,C 180,E1 21706.156,E2 21706.156} C_VEL
LIN {X 0,Y 592.466,Z 1248.815,A -85,B 0,C 180,E1 21703.768,E2 21703.768} C_VEL
LIN {X 0,Y 592.156,Z 1256.91,A -85,B 0,C 180,E1 21701.101,E2 21701.101} C_VEL
LIN {X 0,Y 592.003,Z 1262.622,A -85,B 0,C 180,E1 21698.746,E2 21698.746} C_VEL
LIN {X 0,Y 591.946,Z 1267.106,A -85,B 0,C 180,E1 21696.306,E2 21696.306} C_VEL
LIN {X 0,Y 591.914,Z 1270.301,A -85,B 0,C 180,E1 21693.683,E2 21693.683} C_VEL
LIN {X 0,Y 591.898,Z 1271.703,A -85,B 0,C 180,E1 21691.261,E2 21691.261} C_VEL
LIN {X 0,Y 591.864,Z 1271.838,A -85,B 0,C 180,E1 21689.228,E2 21689.228} C_VEL
LIN {X 0,Y 591.909,Z 1270.981,A -85,B 0,C 180,E1 21687.195,E2 21687.195} C_VEL
LIN {X 0,Y 591.919,Z 1269.057,A -85,B 0,C 180,E1 21685.061,E2 21685.061} C_VEL
LIN {X 0,Y 591.96,Z 1265.667,A -85,B 0,C 180,E1 21682.725,E2 21682.725} C_VEL
LIN {X 0,Y 592.033,Z 1260.469,A -85,B 0,C 180,E1 21680.182,E2 21680.182} C_VEL
LIN {X 0,Y 592.264,Z 1253.805,A -85,B 0,C 180,E1 21677.722,E2 21677.722} C_VEL
LIN {X 0,Y 592.58,Z 1246.683,A -85,B 0,C 180,E1 21675.542,E2 21675.542} C_VEL
LIN {X 0,Y 593.06,Z 1238.688,A -85,B 0,C 180,E1 21673.449,E2 21673.449} C_VEL
LIN {X 0,Y 593.773,Z 1228.514,A -85,B 0,C 180,E1 21671.14,E2 21671.14} C_VEL
LIN {X 0,Y 594.937,Z 1214.99,A -85,B 0,C 180,E1 21668.511,E2 21668.511} C_VEL
LIN {X 0,Y 596.195,Z 1202.394,A -85,B 0,C 180,E1 21666.374,E2 21666.374} C_VEL
LIN {X 0,Y 597.68,Z 1188.904,A -85,B 0,C 180,E1 21664.328,E2 21664.328} C_VEL
LIN {X 0,Y 599.915,Z 1170.341,A -85,B 0,C 180,E1 21661.848,E2 21661.848} C_VEL
LIN {X 0,Y 601.973,Z 1154.048,A -85,B 0,C 180,E1 21659.928,E2 21659.928} C_VEL
LIN {X 0,Y 604.165,Z 1137.706,A -85,B 0,C 180,E1 21658.194,E2 21658.194} C_VEL
LIN {X 0,Y 607.023,Z 1117.034,A -85,B 0,C 180,E1 21656.23,E2 21656.23} C_VEL
LIN {X 0,Y 609.836,Z 1095.8,A -85,B 0,C 180,E1 21654.468,E2 21654.468} C_VEL
LIN {X 0,Y 612.364,Z 1076.938,A -85,B 0,C 180,E1 21653.072,E2 21653.072} C_VEL
LIN {X 0,Y 615.131,Z 1055.804,A -85,B 0,C 180,E1 21651.68,E2 21651.68} C_VEL
LIN {X 0,Y 618.26,Z 1030.528,A -85,B 0,C 180,E1 21650.242,E2 21650.242} C_VEL
LIN {X 0,Y 620.673,Z 1009.158,A -85,B 0,C 180,E1 21649.193,E2 21649.193} C_VEL
LIN {X 0,Y 622.803,Z 988.581,A -85,B 0,C 180,E1 21648.314,E2 21648.314} C_VEL
LIN {X 0,Y 624.703,Z 968.447,A -85,B 0,C 180,E1 21647.573,E2 21647.573} C_VEL
LIN {X 0,Y 626.621,Z 945.459,A -85,B 0,C 180,E1 21646.861,E2 21646.861} C_VEL
LIN {X 0,Y 628.581,Z 916.646,A -85,B 0,C 180,E1 21646.166,E2 21646.166} C_VEL
LIN {X 0,Y 629.728,Z 893.59,A -85,B 0,C 180,E1 21645.754,E2 21645.754} C_VEL
LIN {X 0,Y 634.815,Z 688.505,A -85,B 0,C 180,E1 21642.926,E2 21642.926} C_VEL
LIN {X 0,Y 640.077,Z 484.004,A -85,B 0,C 180,E1 21640.052,E2 21640.052} C_VEL
LIN {X 0,Y 639.985,Z 482.453,A -85,B 0,C 180,E1 21640.015,E2 21640.015} C_VEL
LIN {X 0,Y 628.532,Z 465.508,A -85,B 0,C 180,E1 21638.449,E2 21638.449} C_VEL
LIN {X 0,Y 616.397,Z 448.624,A -85,B 0,C 180,E1 21636.681,E2 21636.681} C_VEL
LIN {X 0,Y 607.96,Z 437.448,A -85,B 0,C 180,E1 21635.375,E2 21635.375} C_VEL
LIN {X 0,Y 600.268,Z 427.651,A -85,B 0,C 180,E1 21634.121,E2 21634.121} C_VEL
LIN {X 0,Y 596.71,Z 423.032,A -85,B 0,C 180,E1 21633.514,E2 21633.514} C_VEL
LIN {X 0,Y 594.231,Z 420.481,A -85,B 0,C 180,E1 21633.095,E2 21633.095} C_VEL
LIN {X 0,Y 593.597,Z 419.169,A -85,B 0,C 180,E1 21632.962,E2 21632.962} C_VEL
LIN {X 0,Y 593.17,Z 417.333,A -85,B 0,C 180,E1 21632.644,E2 21632.644} C_VEL
LIN {X 0,Y 593.136,Z 417.309,A -85,B 0,C 180,E1 21629.488,E2 21629.488} C_VEL
LIN {X 0,Y 593.147,Z 417.318,A -85,B 0,C 180,E1 21626.642,E2 21626.642} C_VEL
LIN {X 0,Y 593.139,Z 417.346,A -85,B 0,C 180,E1 21623.271,E2 21623.271} C_VEL
LIN {X 0,Y 593.141,Z 417.303,A -85,B 0,C 180,E1 21620.416,E2 21620.416} C_VEL
LIN {X 0,Y 593.138,Z 417.344,A -85,B 0,C 180,E1 21617.112,E2 21617.112} C_VEL
LIN {X 0,Y 593.132,Z 417.3,A -85,B 0,C 180,E1 21614.248,E2 21614.248} C_VEL
LIN {X 0,Y 593.136,Z 417.338,A -85,B 0,C 180,E1 21610.883,E2 21610.883} C_VEL
LIN {X 0,Y 593.139,Z 417.307,A -85,B 0,C 180,E1 21607.946,E2 21607.946} C_VEL
LIN {X 0,Y 593.131,Z 417.335,A -85,B 0,C 180,E1 21604.641,E2 21604.641} C_VEL
LIN {X 0,Y 593.137,Z 417.311,A -85,B 0,C 180,E1 21601.699,E2 21601.699} C_VEL
LIN {X 0,Y 593.13,Z 417.333,A -85,B 0,C 180,E1 21598.454,E2 21598.454} C_VEL
LIN {X 0,Y 593.13,Z 417.314,A -85,B 0,C 180,E1 21595.552,E2 21595.552} C_VEL
LIN {X 0,Y 593.128,Z 417.33,A -85,B 0,C 180,E1 21592.249,E2 21592.249} C_VEL
LIN {X 0,Y 593.122,Z 417.318,A -85,B 0,C 180,E1 21589.411,E2 21589.411} C_VEL
LIN {X 0,Y 593.133,Z 417.32,A -85,B 0,C 180,E1 21586.146,E2 21586.146} C_VEL
LIN {X 0,Y 593.112,Z 417.328,A -85,B 0,C 180,E1 21583.346,E2 21583.346} C_VEL
LIN {X 0,Y 593.161,Z 417.301,A -85,B 0,C 180,E1 21580.195,E2 21580.195} C_VEL
LIN {X 0,Y 593.109,Z 417.346,A -85,B 0,C 180,E1 21577.29,E2 21577.29} C_VEL
LIN {X 0,Y 593.178,Z 417.301,A -85,B 0,C 180,E1 21574.221,E2 21574.221} C_VEL
LIN {X 0,Y 593.104,Z 417.33,A -85,B 0,C 180,E1 21571.174,E2 21571.174} C_VEL
LIN {X 0,Y 593.145,Z 417.334,A -85,B 0,C 180,E1 21568.343,E2 21568.343} C_VEL
LIN {X 0,Y 593.21,Z 417.516,A -85,B 0,C 180,E1 21568.044,E2 21568.044} C_VEL
LIN {X 0,Y 594.548,Z 420.997,A -85,B 0,C 180,E1 21567.441,E2 21567.441} C_VEL
LIN {X 0,Y 595.727,Z 422.855,A -85,B 0,C 180,E1 21567.056,E2 21567.056} C_VEL
LIN {X 0,Y 597.833,Z 426.64,A -85,B 0,C 180,E1 21566.356,E2 21566.356} C_VEL
LIN {X 0,Y 601.901,Z 432.044,A -85,B 0,C 180,E1 21565.668,E2 21565.668} C_VEL
LIN {X 0,Y 614.159,Z 448.348,A -85,B 0,C 180,E1 21563.715,E2 21563.715} C_VEL
LIN {X 0,Y 627.623,Z 467.291,A -85,B 0,C 180,E1 21561.732,E2 21561.732} C_VEL
LIN {X 0,Y 640.177,Z 486.019,A -85,B 0,C 180,E1 21560.012,E2 21560.012} C_VEL
LIN {X 0,Y 635.236,Z 679.349,A -85,B 0,C 180,E1 21557.291,E2 21557.291} C_VEL
LIN {X 0,Y 629.875,Z 899.513,A -85,B 0,C 180,E1 21554.261,E2 21554.261} C_VEL
LIN {X 0,Y 628.832,Z 921.641,A -85,B 0,C 180,E1 21553.887,E2 21553.887} C_VEL
LIN {X 0,Y 627.519,Z 942.83,A -85,B 0,C 180,E1 21553.422,E2 21553.422} C_VEL
LIN {X 0,Y 625.854,Z 965.146,A -85,B 0,C 180,E1 21552.811,E2 21552.811} C_VEL
LIN {X 0,Y 623.349,Z 993.25,A -85,B 0,C 180,E1 21551.852,E2 21551.852} C_VEL
LIN {X 0,Y 621.097,Z 1015.408,A -85,B 0,C 180,E1 21550.93,E2 21550.93} C_VEL
LIN {X 0,Y 618.932,Z 1034.753,A -85,B 0,C 180,E1 21550.008,E2 21550.008} C_VEL
LIN {X 0,Y 616.644,Z 1053.8,A -85,B 0,C 180,E1 21548.981,E2 21548.981} C_VEL
LIN {X 0,Y 614.279,Z 1072.493,A -85,B 0,C 180,E1 21547.849,E2 21547.849} C_VEL
LIN {X 0,Y 611.521,Z 1093.716,A -85,B 0,C 180,E1 21546.403,E2 21546.403} C_VEL
LIN {X 0,Y 608.291,Z 1117.261,A -85,B 0,C 180,E1 21544.56,E2 21544.56} C_VEL
LIN {X 0,Y 605.867,Z 1134.981,A -85,B 0,C 180,E1 21542.993,E2 21542.993} C_VEL
LIN {X 0,Y 603.595,Z 1151.857,A -85,B 0,C 180,E1 21541.338,E2 21541.338} C_VEL
LIN {X 0,Y 601.158,Z 1170.765,A -85,B 0,C 180,E1 21539.27,E2 21539.27} C_VEL
LIN {X 0,Y 598.938,Z 1188.101,A -85,B 0,C 180,E1 21537.109,E2 21537.109} C_VEL
LIN {X 0,Y 597.318,Z 1202.109,A -85,B 0,C 180,E1 21535.158,E2 21535.158} C_VEL
LIN {X 0,Y 595.735,Z 1217.201,A -85,B 0,C 180,E1 21532.808,E2 21532.808} C_VEL
LIN {X 0,Y 594.394,Z 1231.258,A -85,B 0,C 180,E1 21530.271,E2 21530.271} C_VEL
LIN {X 0,Y 593.542,Z 1241.546,A -85,B 0,C 180,E1 21528.155,E2 21528.155} C_VEL
LIN {X 0,Y 592.921,Z 1250.938,A -85,B 0,C 180,E1 21525.951,E2 21525.951} C_VEL
LIN {X 0,Y 592.415,Z 1260.622,A -85,B 0,C 180,E1 21523.267,E2 21523.267} C_VEL
LIN {X 0,Y 592.14,Z 1267.298,A -85,B 0,C 180,E1 21520.997,E2 21520.997} C_VEL
LIN {X 0,Y 592.007,Z 1272.729,A -85,B 0,C 180,E1 21518.74,E2 21518.74} C_VEL
LIN {X 0,Y 591.945,Z 1277.19,A -85,B 0,C 180,E1 21516.3,E2 21516.3} C_VEL
LIN {X 0,Y 591.914,Z 1280.337,A -85,B 0,C 180,E1 21513.677,E2 21513.677} C_VEL
LIN {X 0,Y 591.9,Z 1281.692,A -85,B 0,C 180,E1 21511.352,E2 21511.352} C_VEL
LIN {X 0,Y 591.864,Z 1281.849,A -85,B 0,C 180,E1 21509.32,E2 21509.32} C_VEL
LIN {X 0,Y 591.909,Z 1281.013,A -85,B 0,C 180,E1 21507.286,E2 21507.286} C_VEL
LIN {X 0,Y 591.918,Z 1279.111,A -85,B 0,C 180,E1 21505.152,E2 21505.152} C_VEL
LIN {X 0,Y 591.961,Z 1275.743,A -85,B 0,C 180,E1 21502.817,E2 21502.817} C_VEL
LIN {X 0,Y 592.04,Z 1270.338,A -85,B 0,C 180,E1 21500.176,E2 21500.176} C_VEL
LIN {X 0,Y 592.266,Z 1263.649,A -85,B 0,C 180,E1 21497.716,E2 21497.716} C_VEL
LIN {X 0,Y 592.592,Z 1256.502,A -85,B 0,C 180,E1 21495.537,E2 21495.537} C_VEL
LIN {X 0,Y 593.07,Z 1248.484,A -85,B 0,C 180,E1 21493.443,E2 21493.443} C_VEL
LIN {X 0,Y 593.838,Z 1237.82,A -85,B 0,C 180,E1 21491.034,E2 21491.034} C_VEL
LIN {X 0,Y 594.963,Z 1224.712,A -85,B 0,C 180,E1 21488.506,E2 21488.506} C_VEL
LIN {X 0,Y 596.224,Z 1212.087,A -85,B 0,C 180,E1 21486.369,E2 21486.369} C_VEL
LIN {X 0,Y 597.811,Z 1197.851,A -85,B 0,C 180,E1 21484.221,E2 21484.221} C_VEL
LIN {X 0,Y 599.967,Z 1179.897,A -85,B 0,C 180,E1 21481.839,E2 21481.839} C_VEL
LIN {X 0,Y 602.07,Z 1163.355,A -85,B 0,C 180,E1 21479.896,E2 21479.896} C_VEL
LIN {X 0,Y 604.302,Z 1146.732,A -85,B 0,C 180,E1 21478.14,E2 21478.14} C_VEL
LIN {X 0,Y 607.348,Z 1124.345,A -85,B 0,C 180,E1 21476.044,E2 21476.044} C_VEL
LIN {X 0,Y 609.911,Z 1105.196,A -85,B 0,C 180,E1 21474.466,E2 21474.466} C_VEL
LIN {X 0,Y 612.447,Z 1086.279,A -85,B 0,C 180,E1 21473.071,E2 21473.071} C_VEL
LIN {X 0,Y 615.463,Z 1063.469,A -85,B 0,C 180,E1 21471.579,E2 21471.579} C_VEL
LIN {X 0,Y 618.363,Z 1039.667,A -85,B 0,C 180,E1 21470.243,E2 21470.243} C_VEL
LIN {X 0,Y 620.678,Z 1019.126,A -85,B 0,C 180,E1 21469.237,E2 21469.237} C_VEL
LIN {X 0,Y 622.707,Z 999.524,A -85,B 0,C 180,E1 21468.396,E2 21468.396} C_VEL
LIN {X 0,Y 624.669,Z 978.833,A -85,B 0,C 180,E1 21467.632,E2 21467.632} C_VEL
LIN {X 0,Y 626.531,Z 956.552,A -85,B 0,C 180,E1 21466.937,E2 21466.937} C_VEL
LIN {X 0,Y 628.503,Z 928.007,A -85,B 0,C 180,E1 21466.239,E2 21466.239} C_VEL
LIN {X 0,Y 629.706,Z 903.859,A -85,B 0,C 180,E1 21465.804,E2 21465.804} C_VEL
LIN {X 0,Y 634.118,Z 724.94,A -85,B 0,C 180,E1 21463.34,E2 21463.34} C_VEL
LIN {X 0,Y 639.65,Z 506.964,A -85,B 0,C 180,E1 21460.289,E2 21460.289} C_VEL
LIN {X 0,Y 640.071,Z 485.866,A -85,B 0,C 180,E1 21459.974,E2 21459.974} C_VEL
LIN {X 0,Y 625.997,Z 464.845,A -85,B 0,C 180,E1 21458.036,E2 21458.036} C_VEL
LIN {X 0,Y 612.709,Z 446.398,A -85,B 0,C 180,E1 21456.066,E2 21456.066} C_VEL
LIN {X 0,Y 605.25,Z 436.631,A -85,B 0,C 180,E1 21454.891,E2 21454.891} C_VEL
LIN {X 0,Y 601.492,Z 431.608,A -85,B 0,C 180,E1 21454.272,E2 21454.272} C_VEL
LIN {X 0,Y 597.463,Z 426.249,A -85,B 0,C 180,E1 21453.581,E2 21453.581} C_VEL
LIN {X 0,Y 595.706,Z 422.762,A -85,B 0,C 180,E1 21452.939,E2 21452.939} C_VEL
LIN {X 0,Y 593.521,Z 418.829,A -85,B 0,C 180,E1 21452.165,E2 21452.165} C_VEL
LIN {X 0,Y 593.165,Z 417.345,A -85,B 0,C 180,E1 21451.902,E2 21451.902} C_VEL
LIN {X 0,Y 593.114,Z 417.319,A -85,B 0,C 180,E1 21449.047,E2 21449.047} C_VEL
LIN {X 0,Y 593.189,Z 417.303,A -85,B 0,C 180,E1 21445.993,E2 21445.993} C_VEL
LIN {X 0,Y 593.126,Z 417.348,A -85,B 0,C 180,E1 21442.918,E2 21442.918} C_VEL
LIN {X 0,Y 593.197,Z 417.299,A -85,B 0,C 180,E1 21439.853,E2 21439.853} C_VEL
LIN {X 0,Y 593.137,Z 417.338,A -85,B 0,C 180,E1 21436.754,E2 21436.754} C_VEL
LIN {X 0,Y 593.199,Z 417.307,A -85,B 0,C 180,E1 21433.65,E2 21433.65} C_VEL
LIN {X 0,Y 593.146,Z 417.32,A -85,B 0,C 180,E1 21430.49,E2 21430.49} C_VEL
LIN {X 0,Y 593.197,Z 417.323,A -85,B 0,C 180,E1 21427.263,E2 21427.263} C_VEL
LIN {X 0,Y 593.157,Z 417.309,A -85,B 0,C 180,E1 21424.157,E2 21424.157} C_VEL
LIN {X 0,Y 593.183,Z 417.337,A -85,B 0,C 180,E1 21420.869,E2 21420.869} C_VEL
LIN {X 0,Y 593.184,Z 417.298,A -85,B 0,C 180,E1 21417.681,E2 21417.681} C_VEL
LIN {X 0,Y 593.169,Z 417.339,A -85,B 0,C 180,E1 21414.389,E2 21414.389} C_VEL
LIN {X 0,Y 593.187,Z 417.294,A -85,B 0,C 180,E1 21411.274,E2 21411.274} C_VEL
LIN {X 0,Y 593.173,Z 417.342,A -85,B 0,C 180,E1 21408.034,E2 21408.034} C_VEL
LIN {X 0,Y 593.18,Z 417.297,A -85,B 0,C 180,E1 21404.854,E2 21404.854} C_VEL
LIN {X 0,Y 593.185,Z 417.335,A -85,B 0,C 180,E1 21401.625,E2 21401.625} C_VEL
LIN {X 0,Y 593.195,Z 417.314,A -85,B 0,C 180,E1 21398.337,E2 21398.337} C_VEL
LIN {X 0,Y 593.182,Z 417.303,A -85,B 0,C 180,E1 21395.076,E2 21395.076} C_VEL
LIN {X 0,Y 593.194,Z 417.341,A -85,B 0,C 180,E1 21391.833,E2 21391.833} C_VEL
LIN {X 0,Y 593.168,Z 417.319,A -85,B 0,C 180,E1 21388.609,E2 21388.609} C_VEL
LIN {X 0,Y 593.223,Z 417.544,A -85,B 0,C 180,E1 21387.187,E2 21387.187} C_VEL
LIN {X 0,Y 593.96,Z 419.912,A -85,B 0,C 180,E1 21386.859,E2 21386.859} C_VEL
LIN {X 0,Y 596.15,Z 422.608,A -85,B 0,C 180,E1 21386.479,E2 21386.479} C_VEL
LIN {X 0,Y 597.528,Z 423.979,A -85,B 0,C 180,E1 21386.25,E2 21386.25} C_VEL
LIN {X 0,Y 606.9,Z 436.109,A -85,B 0,C 180,E1 21384.699,E2 21384.699} C_VEL
LIN {X 0,Y 610.625,Z 440.958,A -85,B 0,C 180,E1 21384.111,E2 21384.111} C_VEL
LIN {X 0,Y 621.29,Z 455.229,A -85,B 0,C 180,E1 21382.501,E2 21382.501} C_VEL
LIN {X 0,Y 632.209,Z 470.864,A -85,B 0,C 180,E1 21380.947,E2 21380.947} C_VEL
LIN {X 0,Y 640.113,Z 482.673,A -85,B 0,C 180,E1 21379.877,E2 21379.877} C_VEL
LIN {X 0,Y 635.701,Z 653.001,A -85,B 0,C 180,E1 21377.478,E2 21377.478} C_VEL
LIN {X 0,Y 634.831,Z 660.704,A -85,B 0,C 180,E1 21377.437,E2 21377.437} C_VEL
LIN {X 0,Y 630.073,Z 681.362,A -85,B 0,C 180,E1 21377.569,E2 21377.569} C_VEL
LIN {X 0,Y 629.384,Z 687.971,A -85,B 0,C 180,E1 21377.528,E2 21377.528} C_VEL
LIN {X 0,Y 624.027,Z 893.124,A -85,B 0,C 180,E1 21374.678,E2 21374.678} C_VEL
LIN {X 0,Y 622.864,Z 915.669,A -85,B 0,C 180,E1 21374.277,E2 21374.277} C_VEL
LIN {X 0,Y 621.034,Z 942.554,A -85,B 0,C 180,E1 21373.643,E2 21373.643} C_VEL
LIN {X 0,Y 618.881,Z 967.082,A -85,B 0,C 180,E1 21372.891,E2 21372.891} C_VEL
LIN {X 0,Y 616.867,Z 987.314,A -85,B 0,C 180,E1 21372.15,E2 21372.15} C_VEL
LIN {X 0,Y 614.786,Z 1006.719,A -85,B 0,C 180,E1 21371.325,E2 21371.325} C_VEL
LIN {X 0,Y 612.65,Z 1024.808,A -85,B 0,C 180,E1 21370.455,E2 21370.455} C_VEL
LIN {X 0,Y 610.226,Z 1043.927,A -85,B 0,C 180,E1 21369.417,E2 21369.417} C_VEL
LIN {X 0,Y 607.628,Z 1063.403,A -85,B 0,C 180,E1 21368.225,E2 21368.225} C_VEL
LIN {X 0,Y 604.453,Z 1086.604,A -85,B 0,C 180,E1 21366.616,E2 21366.616} C_VEL
LIN {X 0,Y 601.301,Z 1108.112,A -85,B 0,C 180,E1 21364.893,E2 21364.893} C_VEL
LIN {X 0,Y 598.768,Z 1125.59,A -85,B 0,C 180,E1 21363.327,E2 21363.327} C_VEL
LIN {X 0,Y 596.363,Z 1142.408,A -85,B 0,C 180,E1 21361.656,E2 21361.656} C_VEL
LIN {X 0,Y 593.53,Z 1162.931,A -85,B 0,C 180,E1 21359.357,E2 21359.357} C_VEL
LIN {X 0,Y 591.427,Z 1178.506,A -85,B 0,C 180,E1 21357.379,E2 21357.379} C_VEL
LIN {X 0,Y 589.69,Z 1192.475,A -85,B 0,C 180,E1 21355.405,E2 21355.405} C_VEL
LIN {X 0,Y 587.94,Z 1208.117,A -85,B 0,C 180,E1 21352.922,E2 21352.922} C_VEL
LIN {X 0,Y 586.57,Z 1221.523,A -85,B 0,C 180,E1 21350.456,E2 21350.456} C_VEL
LIN {X 0,Y 585.657,Z 1231.779,A -85,B 0,C 180,E1 21348.311,E2 21348.311} C_VEL
LIN {X 0,Y 584.974,Z 1241.543,A -85,B 0,C 180,E1 21345.976,E2 21345.976} C_VEL
LIN {X 0,Y 584.43,Z 1251.184,A -85,B 0,C 180,E1 21343.221,E2 21343.221} C_VEL
LIN {X 0,Y 584.152,Z 1257.68,A -85,B 0,C 180,E1 21340.955,E2 21340.955} C_VEL
LIN {X 0,Y 584.012,Z 1263.033,A -85,B 0,C 180,E1 21338.668,E2 21338.668} C_VEL
LIN {X 0,Y 583.941,Z 1267.562,A -85,B 0,C 180,E1 21336.097,E2 21336.097} C_VEL
LIN {X 0,Y 583.913,Z 1270.438,A -85,B 0,C 180,E1 21333.537,E2 21333.537} C_VEL
LIN {X 0,Y 583.899,Z 1271.703,A -85,B 0,C 180,E1 21331.278,E2 21331.278} C_VEL
LIN {X 0,Y 583.864,Z 1271.838,A -85,B 0,C 180,E1 21329.218,E2 21329.218} C_VEL
LIN {X 0,Y 583.91,Z 1270.981,A -85,B 0,C 180,E1 21327.157,E2 21327.157} C_VEL
LIN {X 0,Y 583.92,Z 1269.054,A -85,B 0,C 180,E1 21324.993,E2 21324.993} C_VEL
LIN {X 0,Y 583.958,Z 1265.663,A -85,B 0,C 180,E1 21322.625,E2 21322.625} C_VEL
LIN {X 0,Y 584.057,Z 1260.467,A -85,B 0,C 180,E1 21320.046,E2 21320.046} C_VEL
LIN {X 0,Y 584.298,Z 1253.803,A -85,B 0,C 180,E1 21317.552,E2 21317.552} C_VEL
LIN {X 0,Y 584.655,Z 1246.68,A -85,B 0,C 180,E1 21315.342,E2 21315.342} C_VEL
LIN {X 0,Y 585.152,Z 1238.684,A -85,B 0,C 180,E1 21313.219,E2 21313.219} C_VEL
LIN {X 0,Y 585.893,Z 1228.978,A -85,B 0,C 180,E1 21310.98,E2 21310.98} C_VEL
LIN {X 0,Y 587.131,Z 1215.557,A -85,B 0,C 180,E1 21308.316,E2 21308.316} C_VEL
LIN {X 0,Y 588.456,Z 1203.023,A -85,B 0,C 180,E1 21306.151,E2 21306.151} C_VEL
LIN {X 0,Y 590.041,Z 1189.598,A -85,B 0,C 180,E1 21304.078,E2 21304.078} C_VEL
LIN {X 0,Y 592.296,Z 1172.126,A -85,B 0,C 180,E1 21301.686,E2 21301.686} C_VEL
LIN {X 0,Y 594.63,Z 1154.705,A -85,B 0,C 180,E1 21299.598,E2 21299.598} C_VEL
LIN {X 0,Y 596.86,Z 1138.958,A -85,B 0,C 180,E1 21297.899,E2 21297.899} C_VEL
LIN {X 0,Y 599.538,Z 1120.556,A -85,B 0,C 180,E1 21296.111,E2 21296.111} C_VEL
LIN {X 0,Y 602.785,Z 1097.793,A -85,B 0,C 180,E1 21294.164,E2 21294.164} C_VEL
LIN {X 0,Y 605.528,Z 1078.395,A -85,B 0,C 180,E1 21292.704,E2 21292.704} C_VEL
LIN {X 0,Y 608.197,Z 1059.038,A -85,B 0,C 180,E1 21291.404,E2 21291.404} C_VEL
LIN {X 0,Y 611.355,Z 1035.455,A -85,B 0,C 180,E1 21290.008,E2 21290.008} C_VEL
LIN {X 0,Y 614.334,Z 1010.586,A -85,B 0,C 180,E1 21288.76,E2 21288.76} C_VEL
LIN {X 0,Y 616.523,Z 990.592,A -85,B 0,C 180,E1 21287.891,E2 21287.891} C_VEL
LIN {X 0,Y 618.58,Z 970.093,A -85,B 0,C 180,E1 21287.122,E2 21287.122} C_VEL
LIN {X 0,Y 620.44,Z 949.136,A -85,B 0,C 180,E1 21286.457,E2 21286.457} C_VEL
LIN {X 0,Y 622.258,Z 925.399,A -85,B 0,C 180,E1 21285.841,E2 21285.841} C_VEL
LIN {X 0,Y 623.883,Z 896.631,A -85,B 0,C 180,E1 21285.285,E2 21285.285} C_VEL
LIN {X 0,Y 625.65,Z 833.91,A -85,B 0,C 180,E1 21284.404,E2 21284.404} C_VEL
LIN {X 0,Y 631.347,Z 614.091,A -85,B 0,C 180,E1 21281.345,E2 21281.345} C_VEL
LIN {X 0,Y 634.786,Z 486.411,A -85,B 0,C 180,E1 21279.522,E2 21279.522} C_VEL
LIN {X 0,Y 620.345,Z 465.184,A -85,B 0,C 180,E1 21277.479,E2 21277.479} C_VEL
LIN {X 0,Y 609.181,Z 449.953,A -85,B 0,C 180,E1 21275.785,E2 21275.785} C_VEL
LIN {X 0,Y 600.687,Z 438.766,A -85,B 0,C 180,E1 21274.411,E2 21274.411} C_VEL
LIN {X 0,Y 593.668,Z 429.935,A -85,B 0,C 180,E1 21273.217,E2 21273.217} C_VEL
LIN {X 0,Y 590.879,Z 426.681,A -85,B 0,C 180,E1 21272.729,E2 21272.729} C_VEL
LIN {X 0,Y 589.497,Z 424.434,A -85,B 0,C 180,E1 21272.469,E2 21272.469} C_VEL
LIN {X 0,Y 586.687,Z 422.013,A -85,B 0,C 180,E1 21271.979,E2 21271.979} C_VEL
LIN {X 0,Y 585.374,Z 419.212,A -85,B 0,C 180,E1 21271.685,E2 21271.685} C_VEL
LIN {X 0,Y 585.199,Z 418.313,A -85,B 0,C 180,E1 21271.514,E2 21271.514} C_VEL
LIN {X 0,Y 585.22,Z 418.314,A -85,B 0,C 180,E1 21268.581,E2 21268.581} C_VEL
LIN {X 0,Y 585.193,Z 418.29,A -85,B 0,C 180,E1 21265.288,E2 21265.288} C_VEL
LIN {X 0,Y 585.225,Z 418.326,A -85,B 0,C 180,E1 21262.29,E2 21262.29} C_VEL
LIN {X 0,Y 585.192,Z 418.307,A -85,B 0,C 180,E1 21259.048,E2 21259.048} C_VEL
LIN {X 0,Y 585.21,Z 418.306,A -85,B 0,C 180,E1 21256.171,E2 21256.171} C_VEL
LIN {X 0,Y 585.195,Z 418.32,A -85,B 0,C 180,E1 21252.934,E2 21252.934} C_VEL
LIN {X 0,Y 585.199,Z 418.299,A -85,B 0,C 180,E1 21250.037,E2 21250.037} C_VEL
LIN {X 0,Y 585.191,Z 418.332,A -85,B 0,C 180,E1 21246.672,E2 21246.672} C_VEL
LIN {X 0,Y 585.196,Z 418.296,A -85,B 0,C 180,E1 21243.821,E2 21243.821} C_VEL
LIN {X 0,Y 585.191,Z 418.334,A -85,B 0,C 180,E1 21240.49,E2 21240.49} C_VEL
LIN {X 0,Y 585.19,Z 418.296,A -85,B 0,C 180,E1 21237.65,E2 21237.65} C_VEL
LIN {X 0,Y 585.192,Z 418.335,A -85,B 0,C 180,E1 21234.313,E2 21234.313} C_VEL
LIN {X 0,Y 585.18,Z 418.298,A -85,B 0,C 180,E1 21231.55,E2 21231.55} C_VEL
LIN {X 0,Y 585.199,Z 418.335,A -85,B 0,C 180,E1 21228.223,E2 21228.223} C_VEL
LIN {X 0,Y 585.169,Z 418.295,A -85,B 0,C 180,E1 21225.452,E2 21225.452} C_VEL
LIN {X 0,Y 585.231,Z 418.332,A -85,B 0,C 180,E1 21222.295,E2 21222.295} C_VEL
LIN {X 0,Y 585.166,Z 418.289,A -85,B 0,C 180,E1 21219.286,E2 21219.286} C_VEL
LIN {X 0,Y 585.244,Z 418.318,A -85,B 0,C 180,E1 21216.221,E2 21216.221} C_VEL
LIN {X 0,Y 585.166,Z 418.317,A -85,B 0,C 180,E1 21213.076,E2 21213.076} C_VEL
LIN {X 0,Y 585.238,Z 418.29,A -85,B 0,C 180,E1 21209.96,E2 21209.96} C_VEL
LIN {X 0,Y 585.182,Z 418.448,A -85,B 0,C 180,E1 21209.194,E2 21209.194} C_VEL
LIN {X 0,Y 586.556,Z 421.9,A -85,B 0,C 180,E1 21208.558,E2 21208.558} C_VEL
LIN {X 0,Y 587.812,Z 423.476,A -85,B 0,C 180,E1 21208.175,E2 21208.175} C_VEL
LIN {X 0,Y 589.233,Z 426.705,A -85,B 0,C 180,E1 21207.63,E2 21207.63} C_VEL
LIN {X 0,Y 591.973,Z 430.229,A -85,B 0,C 180,E1 21207.138,E2 21207.138} C_VEL
LIN {X 0,Y 595.748,Z 434.83,A -85,B 0,C 180,E1 21206.483,E2 21206.483} C_VEL
LIN {X 0,Y 607.172,Z 449.956,A -85,B 0,C 180,E1 21204.589,E2 21204.589} C_VEL
LIN {X 0,Y 618.446,Z 465.612,A -85,B 0,C 180,E1 21202.852,E2 21202.852} C_VEL
LIN {X 0,Y 627.451,Z 478.754,A -85,B 0,C 180,E1 21201.545,E2 21201.545} C_VEL
LIN {X 0,Y 634.929,Z 490.133,A -85,B 0,C 180,E1 21200.507,E2 21200.507} C_VEL
LIN {X 0,Y 629.537,Z 689.636,A -85,B 0,C 180,E1 21197.684,E2 21197.684} C_VEL
LIN {X 0,Y 624.048,Z 901.806,A -85,B 0,C 180,E1 21194.74,E2 21194.74} C_VEL
LIN {X 0,Y 622.935,Z 923.659,A -85,B 0,C 180,E1 21194.359,E2 21194.359} C_VEL
LIN {X 0,Y 621.395,Z 946.888,A -85,B 0,C 180,E1 21193.831,E2 21193.831} C_VEL
LIN {X 0,Y 619.043,Z 975.256,A -85,B 0,C 180,E1 21192.996,E2 21192.996} C_VEL
LIN {X 0,Y 616.898,Z 997.019,A -85,B 0,C 180,E1 21192.207,E2 21192.207} C_VEL
LIN {X 0,Y 614.675,Z 1017.665,A -85,B 0,C 180,E1 21191.327,E2 21191.327} C_VEL
LIN {X 0,Y 612.534,Z 1035.753,A -85,B 0,C 180,E1 21190.451,E2 21190.451} C_VEL
LIN {X 0,Y 610.131,Z 1054.697,A -85,B 0,C 180,E1 21189.417,E2 21189.417} C_VEL
LIN {X 0,Y 607.439,Z 1074.924,A -85,B 0,C 180,E1 21188.172,E2 21188.172} C_VEL
LIN {X 0,Y 603.997,Z 1099.554,A -85,B 0,C 180,E1 21186.433,E2 21186.433} C_VEL
LIN {X 0,Y 601.219,Z 1118.657,A -85,B 0,C 180,E1 21184.892,E2 21184.892} C_VEL
LIN {X 0,Y 598.695,Z 1136.09,A -85,B 0,C 180,E1 21183.325,E2 21183.325} C_VEL
LIN {X 0,Y 596.097,Z 1154.39,A -85,B 0,C 180,E1 21181.496,E2 21181.496} C_VEL
LIN {X 0,Y 593.358,Z 1174.173,A -85,B 0,C 180,E1 21179.25,E2 21179.25} C_VEL
LIN {X 0,Y 591.27,Z 1189.64,A -85,B 0,C 180,E1 21177.272,E2 21177.272} C_VEL
LIN {X 0,Y 589.5,Z 1204.209,A -85,B 0,C 180,E1 21175.193,E2 21175.193} C_VEL
LIN {X 0,Y 587.643,Z 1220.724,A -85,B 0,C 180,E1 21172.506,E2 21172.506} C_VEL
LIN {X 0,Y 586.494,Z 1232.352,A -85,B 0,C 180,E1 21170.335,E2 21170.335} C_VEL
LIN {X 0,Y 585.609,Z 1242.462,A -85,B 0,C 180,E1 21168.204,E2 21168.204} C_VEL
LIN {X 0,Y 584.863,Z 1253.318,A -85,B 0,C 180,E1 21165.566,E2 21165.566} C_VEL
LIN {X 0,Y 584.406,Z 1261.847,A -85,B 0,C 180,E1 21163.049,E2 21163.049} C_VEL
LIN {X 0,Y 584.145,Z 1267.81,A -85,B 0,C 180,E1 21160.949,E2 21160.949} C_VEL
LIN {X 0,Y 584.013,Z 1273.139,A -85,B 0,C 180,E1 21158.662,E2 21158.662} C_VEL
LIN {X 0,Y 583.941,Z 1277.639,A -85,B 0,C 180,E1 21156.091,E2 21156.091} C_VEL
LIN {X 0,Y 583.913,Z 1280.473,A -85,B 0,C 180,E1 21153.531,E2 21153.531} C_VEL
LIN {X 0,Y 583.894,Z 1281.714,A -85,B 0,C 180,E1 21151.273,E2 21151.273} C_VEL
LIN {X 0,Y 583.865,Z 1281.826,A -85,B 0,C 180,E1 21149.212,E2 21149.212} C_VEL
LIN {X 0,Y 583.909,Z 1281.013,A -85,B 0,C 180,E1 21147.249,E2 21147.249} C_VEL
LIN {X 0,Y 583.919,Z 1279.108,A -85,B 0,C 180,E1 21145.086,E2 21145.086} C_VEL
LIN {X 0,Y 583.959,Z 1275.74,A -85,B 0,C 180,E1 21142.718,E2 21142.718} C_VEL
LIN {X 0,Y 584.05,Z 1270.589,A -85,B 0,C 180,E1 21140.14,E2 21140.14} C_VEL
LIN {X 0,Y 584.302,Z 1263.648,A -85,B 0,C 180,E1 21137.546,E2 21137.546} C_VEL
LIN {X 0,Y 584.667,Z 1256.501,A -85,B 0,C 180,E1 21135.336,E2 21135.336} C_VEL
LIN {X 0,Y 585.164,Z 1248.483,A -85,B 0,C 180,E1 21133.213,E2 21133.213} C_VEL
LIN {X 0,Y 585.963,Z 1238.287,A -85,B 0,C 180,E1 21130.873,E2 21130.873} C_VEL
LIN {X 0,Y 587.215,Z 1224.71,A -85,B 0,C 180,E1 21128.208,E2 21128.208} C_VEL
LIN {X 0,Y 588.537,Z 1212.251,A -85,B 0,C 180,E1 21126.069,E2 21126.069} C_VEL
LIN {X 0,Y 590.179,Z 1198.564,A -85,B 0,C 180,E1 21123.971,E2 21123.971} C_VEL
LIN {X 0,Y 592.542,Z 1180.04,A -85,B 0,C 180,E1 21121.473,E2 21121.473} C_VEL
LIN {X 0,Y 594.763,Z 1163.816,A -85,B 0,C 180,E1 21119.543,E2 21119.543} C_VEL
LIN {X 0,Y 597.039,Z 1147.745,A -85,B 0,C 180,E1 21117.819,E2 21117.819} C_VEL
LIN {X 0,Y 600.06,Z 1127.088,A -85,B 0,C 180,E1 21115.836,E2 21115.836} C_VEL
LIN {X 0,Y 603.043,Z 1105.861,A -85,B 0,C 180,E1 21114.057,E2 21114.057} C_VEL
LIN {X 0,Y 605.717,Z 1087.01,A -85,B 0,C 180,E1 21112.651,E2 21112.651} C_VEL
LIN {X 0,Y 608.509,Z 1066.818,A -85,B 0,C 180,E1 21111.308,E2 21111.308} C_VEL
LIN {X 0,Y 611.945,Z 1040.668,A -85,B 0,C 180,E1 21109.802,E2 21109.802} C_VEL
LIN {X 0,Y 614.427,Z 1019.799,A -85,B 0,C 180,E1 21108.769,E2 21108.769} C_VEL
LIN {X 0,Y 616.635,Z 999.521,A -85,B 0,C 180,E1 21107.893,E2 21107.893} C_VEL
LIN {X 0,Y 618.691,Z 978.793,A -85,B 0,C 180,E1 21107.125,E2 21107.125} C_VEL
LIN {X 0,Y 620.64,Z 956.431,A -85,B 0,C 180,E1 21106.426,E2 21106.426} C_VEL
LIN {X 0,Y 622.715,Z 927.787,A -85,B 0,C 180,E1 21105.723,E2 21105.723} C_VEL
LIN {X 0,Y 623.968,Z 903.771,A -85,B 0,C 180,E1 21105.29,E2 21105.29} C_VEL
LIN {X 0,Y 628.6,Z 725.825,A -85,B 0,C 180,E1 21102.821,E2 21102.821} C_VEL
LIN {X 0,Y 634.44,Z 508.061,A -85,B 0,C 180,E1 21099.751,E2 21099.751} C_VEL
LIN {X 0,Y 634.781,Z 489.697,A -85,B 0,C 180,E1 21099.469,E2 21099.469} C_VEL
LIN {X 0,Y 620.301,Z 468.25,A -85,B 0,C 180,E1 21097.424,E2 21097.424} C_VEL
LIN {X 0,Y 609.019,Z 452.488,A -85,B 0,C 180,E1 21095.709,E2 21095.709} C_VEL
LIN {X 0,Y 601.89,Z 443.056,A -85,B 0,C 180,E1 21094.564,E2 21094.564} C_VEL
LIN {X 0,Y 597.914,Z 437.784,A -85,B 0,C 180,E1 21093.898,E2 21093.898} C_VEL
LIN {X 0,Y 594.254,Z 432.91,A -85,B 0,C 180,E1 21093.266,E2 21093.266} C_VEL
LIN {X 0,Y 588.634,Z 425.753,A -85,B 0,C 180,E1 21092.227,E2 21092.227} C_VEL
LIN {X 0,Y 587.492,Z 423.003,A -85,B 0,C 180,E1 21091.73,E2 21091.73} C_VEL
LIN {X 0,Y 585.528,Z 419.867,A -85,B 0,C 180,E1 21091.046,E2 21091.046} C_VEL
LIN {X 0,Y 585.185,Z 418.303,A -85,B 0,C 180,E1 21090.775,E2 21090.775} C_VEL
LIN {X 0,Y 585.199,Z 418.337,A -85,B 0,C 180,E1 21087.473,E2 21087.473} C_VEL
LIN {X 0,Y 585.201,Z 418.297,A -85,B 0,C 180,E1 21084.532,E2 21084.532} C_VEL
LIN {X 0,Y 585.2,Z 418.301,A -85,B 0,C 180,E1 21081.237,E2 21081.237} C_VEL
LIN {X 0,Y 585.23,Z 418.325,A -85,B 0,C 180,E1 21078.204,E2 21078.204} C_VEL
LIN {X 0,Y 585.198,Z 418.286,A -85,B 0,C 180,E1 21074.952,E2 21074.952} C_VEL
LIN {X 0,Y 585.256,Z 418.331,A -85,B 0,C 180,E1 21071.83,E2 21071.83} C_VEL
LIN {X 0,Y 585.205,Z 418.285,A -85,B 0,C 180,E1 21068.648,E2 21068.648} C_VEL
LIN {X 0,Y 585.261,Z 418.323,A -85,B 0,C 180,E1 21065.49,E2 21065.49} C_VEL
LIN {X 0,Y 585.214,Z 418.288,A -85,B 0,C 180,E1 21062.252,E2 21062.252} C_VEL
LIN {X 0,Y 585.257,Z 418.319,A -85,B 0,C 180,E1 21059.021,E2 21059.021} C_VEL
LIN {X 0,Y 585.244,Z 418.295,A -85,B 0,C 180,E1 21055.689,E2 21055.689} C_VEL
LIN {X 0,Y 585.235,Z 418.308,A -85,B 0,C 180,E1 21052.44,E2 21052.44} C_VEL
LIN {X 0,Y 585.248,Z 418.308,A -85,B 0,C 180,E1 21049.168,E2 21049.168} C_VEL
LIN {X 0,Y 585.232,Z 418.293,A -85,B 0,C 180,E1 21045.959,E2 21045.959} C_VEL
LIN {X 0,Y 585.249,Z 418.33,A -85,B 0,C 180,E1 21042.706,E2 21042.706} C_VEL
LIN {X 0,Y 585.25,Z 418.285,A -85,B 0,C 180,E1 21039.393,E2 21039.393} C_VEL
LIN {X 0,Y 585.253,Z 418.313,A -85,B 0,C 180,E1 21036.07,E2 21036.07} C_VEL
LIN {X 0,Y 585.237,Z 418.319,A -85,B 0,C 180,E1 21032.749,E2 21032.749} C_VEL
LIN {X 0,Y 585.247,Z 418.289,A -85,B 0,C 180,E1 21029.508,E2 21029.508} C_VEL
LIN {X 0,Y 585.249,Z 418.435,A -85,B 0,C 180,E1 21028.33,E2 21028.33} C_VEL
LIN {X 0,Y 585.696,Z 420.151,A -85,B 0,C 180,E1 21028.119,E2 21028.119} C_VEL
LIN {X 0,Y 587.603,Z 423.062,A -85,B 0,C 180,E1 21027.754,E2 21027.754} C_VEL
LIN {X 0,Y 590.04,Z 425.106,A -85,B 0,C 180,E1 21027.334,E2 21027.334} C_VEL
LIN {X 0,Y 592.746,Z 429.073,A -85,B 0,C 180,E1 21026.84,E2 21026.84} C_VEL
LIN {X 0,Y 595.095,Z 431.57,A -85,B 0,C 180,E1 21026.441,E2 21026.441} C_VEL
LIN {X 0,Y 606.592,Z 446.396,A -85,B 0,C 180,E1 21024.533,E2 21024.533} C_VEL
LIN {X 0,Y 618.968,Z 463.287,A -85,B 0,C 180,E1 21022.631,E2 21022.631} C_VEL
LIN {X 0,Y 633.12,Z 483.775,A -85,B 0,C 180,E1 21020.618,E2 21020.618} C_VEL
LIN {X 0,Y 634.855,Z 486.791,A -85,B 0,C 180,E1 21020.374,E2 21020.374} C_VEL
LIN {X 0,Y 629.384,Z 687.971,A -85,B 0,C 180,E1 21017.528,E2 21017.528} C_VEL
LIN {X 0,Y 628.51,Z 695.672,A -85,B 0,C 180,E1 21017.487,E2 21017.487} C_VEL
LIN {X 0,Y 623.755,Z 716.326,A -85,B 0,C 180,E1 21017.621,E2 21017.621} C_VEL
LIN {X 0,Y 623.038,Z 722.937,A -85,B 0,C 180,E1 21017.582,E2 21017.582} C_VEL
LIN {X 0,Y 618.313,Z 894.146,A -85,B 0,C 180,E1 21015.186,E2 21015.186} C_VEL
LIN {X 0,Y 617,Z 918.245,A -85,B 0,C 180,E1 21014.748,E2 21014.748} C_VEL
LIN {X 0,Y 614.835,Z 946.703,A -85,B 0,C 180,E1 21014.045,E2 21014.045} C_VEL
LIN {X 0,Y 612.822,Z 968.666,A -85,B 0,C 180,E1 21013.355,E2 21013.355} C_VEL
LIN {X 0,Y 610.721,Z 988.7,A -85,B 0,C 180,E1 21012.61,E2 21012.61} C_VEL
LIN {X 0,Y 608.401,Z 1009.028,A -85,B 0,C 180,E1 21011.73,E2 21011.73} C_VEL
LIN {X 0,Y 605.864,Z 1029.252,A -85,B 0,C 180,E1 21010.728,E2 21010.728} C_VEL
LIN {X 0,Y 602.575,Z 1053.68,A -85,B 0,C 180,E1 21009.338,E2 21009.338} C_VEL
LIN {X 0,Y 599.334,Z 1075.727,A -85,B 0,C 180,E1 21007.877,E2 21007.877} C_VEL
LIN {X 0,Y 596.598,Z 1094.02,A -85,B 0,C 180,E1 21006.512,E2 21006.512} C_VEL
LIN {X 0,Y 593.803,Z 1112.375,A -85,B 0,C 180,E1 21004.986,E2 21004.986} C_VEL
LIN {X 0,Y 590.578,Z 1133.8,A -85,B 0,C 180,E1 21002.98,E2 21002.98} C_VEL
LIN {X 0,Y 587.814,Z 1152.06,A -85,B 0,C 180,E1 21001.027,E2 21001.027} C_VEL
LIN {X 0,Y 585.594,Z 1167.164,A -85,B 0,C 180,E1 20999.233,E2 20999.233} C_VEL
LIN {X 0,Y 583.406,Z 1182.684,A -85,B 0,C 180,E1 20997.188,E2 20997.188} C_VEL
LIN {X 0,Y 581.194,Z 1199.914,A -85,B 0,C 180,E1 20994.605,E2 20994.605} C_VEL
LIN {X 0,Y 579.696,Z 1212.781,A -85,B 0,C 180,E1 20992.403,E2 20992.403} C_VEL
LIN {X 0,Y 578.493,Z 1224.613,A -85,B 0,C 180,E1 20990.12,E2 20990.12} C_VEL
LIN {X 0,Y 577.379,Z 1237.08,A -85,B 0,C 180,E1 20987.332,E2 20987.332} C_VEL
LIN {X 0,Y 576.779,Z 1245.993,A -85,B 0,C 180,E1 20984.972,E2 20984.972} C_VEL
LIN {X 0,Y 576.367,Z 1253.211,A -85,B 0,C 180,E1 20982.73,E2 20982.73} C_VEL
LIN {X 0,Y 576.13,Z 1259.461,A -85,B 0,C 180,E1 20980.401,E2 20980.401} C_VEL
LIN {X 0,Y 575.948,Z 1265.169,A -85,B 0,C 180,E1 20977.685,E2 20977.685} C_VEL
LIN {X 0,Y 575.923,Z 1268.827,A -85,B 0,C 180,E1 20975.182,E2 20975.182} C_VEL
LIN {X 0,Y 575.91,Z 1270.846,A -85,B 0,C 180,E1 20972.988,E2 20972.988} C_VEL
LIN {X 0,Y 575.879,Z 1271.771,A -85,B 0,C 180,E1 20970.998,E2 20970.998} C_VEL
LIN {X 0,Y 575.872,Z 1271.792,A -85,B 0,C 180,E1 20969.008,E2 20969.008} C_VEL
LIN {X 0,Y 575.911,Z 1270.912,A -85,B 0,C 180,E1 20967.017,E2 20967.017} C_VEL
LIN {X 0,Y 575.922,Z 1268.937,A -85,B 0,C 180,E1 20964.823,E2 20964.823} C_VEL
LIN {X 0,Y 575.952,Z 1265.333,A -85,B 0,C 180,E1 20962.321,E2 20962.321} C_VEL
LIN {X 0,Y 576.122,Z 1259.702,A -85,B 0,C 180,E1 20959.605,E2 20959.605} C_VEL
LIN {X 0,Y 576.355,Z 1253.497,A -85,B 0,C 180,E1 20957.275,E2 20957.275} C_VEL
LIN {X 0,Y 576.757,Z 1246.324,A -85,B 0,C 180,E1 20955.034,E2 20955.034} C_VEL
LIN {X 0,Y 577.32,Z 1237.869,A -85,B 0,C 180,E1 20952.777,E2 20952.777} C_VEL
LIN {X 0,Y 578.36,Z 1226.107,A -85,B 0,C 180,E1 20950.092,E2 20950.092} C_VEL
LIN {X 0,Y 579.577,Z 1213.831,A -85,B 0,C 180,E1 20947.699,E2 20947.699} C_VEL
LIN {X 0,Y 580.988,Z 1201.487,A -85,B 0,C 180,E1 20945.564,E2 20945.564} C_VEL
LIN {X 0,Y 582.999,Z 1186.056,A -85,B 0,C 180,E1 20943.193,E2 20943.193} C_VEL
LIN {X 0,Y 585.361,Z 1168.737,A -85,B 0,C 180,E1 20940.873,E2 20940.873} C_VEL
LIN {X 0,Y 587.584,Z 1153.565,A -85,B 0,C 180,E1 20939.055,E2 20939.055} C_VEL
LIN {X 0,Y 590.038,Z 1137.183,A -85,B 0,C 180,E1 20937.282,E2 20937.282} C_VEL
LIN {X 0,Y 593.308,Z 1115.81,A -85,B 0,C 180,E1 20935.223,E2 20935.223} C_VEL
LIN {X 0,Y 596.327,Z 1095.778,A -85,B 0,C 180,E1 20933.535,E2 20933.535} C_VEL
LIN {X 0,Y 599.129,Z 1077.086,A -85,B 0,C 180,E1 20932.129,E2 20932.129} C_VEL
LIN {X 0,Y 601.993,Z 1057.401,A -85,B 0,C 180,E1 20930.808,E2 20930.808} C_VEL
LIN {X 0,Y 605.583,Z 1031.5,A -85,B 0,C 180,E1 20929.299,E2 20929.299} C_VEL
LIN {X 0,Y 608.326,Z 1009.633,A -85,B 0,C 180,E1 20928.208,E2 20928.208} C_VEL
LIN {X 0,Y 610.648,Z 989.375,A -85,B 0,C 180,E1 20927.327,E2 20927.327} C_VEL
LIN {X 0,Y 612.808,Z 968.796,A -85,B 0,C 180,E1 20926.56,E2 20926.56} C_VEL
LIN {X 0,Y 614.833,Z 946.7,A -85,B 0,C 180,E1 20925.865,E2 20925.865} C_VEL
LIN {X 0,Y 616.996,Z 918.217,A -85,B 0,C 180,E1 20925.161,E2 20925.161} C_VEL
LIN {X 0,Y 618.309,Z 894.169,A -85,B 0,C 180,E1 20924.724,E2 20924.724} C_VEL
LIN {X 0,Y 623.134,Z 719.369,A -85,B 0,C 180,E1 20922.278,E2 20922.278} C_VEL
LIN {X 0,Y 629.243,Z 504.586,A -85,B 0,C 180,E1 20919.227,E2 20919.227} C_VEL
LIN {X 0,Y 629.534,Z 490.277,A -85,B 0,C 180,E1 20919.006,E2 20919.006} C_VEL
LIN {X 0,Y 615.781,Z 470.129,A -85,B 0,C 180,E1 20917.015,E2 20917.015} C_VEL
LIN {X 0,Y 605.52,Z 456.051,A -85,B 0,C 180,E1 20915.423,E2 20915.423} C_VEL
LIN {X 0,Y 597.239,Z 445.056,A -85,B 0,C 180,E1 20914.057,E2 20914.057} C_VEL
LIN {X 0,Y 590.774,Z 436.876,A -85,B 0,C 180,E1 20912.937,E2 20912.937} C_VEL
LIN {X 0,Y 587.551,Z 432.88,A -85,B 0,C 180,E1 20912.359,E2 20912.359} C_VEL
LIN {X 0,Y 586.626,Z 431.524,A -85,B 0,C 180,E1 20912.185,E2 20912.185} C_VEL
LIN {X 0,Y 583.52,Z 428.418,A -85,B 0,C 180,E1 20911.624,E2 20911.624} C_VEL
LIN {X 0,Y 581.987,Z 425.638,A -85,B 0,C 180,E1 20911.313,E2 20911.313} C_VEL
LIN {X 0,Y 579.009,Z 423.352,A -85,B 0,C 180,E1 20910.77,E2 20910.77} C_VEL
LIN {X 0,Y 577.528,Z 420.41,A -85,B 0,C 180,E1 20910.451,E2 20910.451} C_VEL
LIN {X 0,Y 577.315,Z 419.271,A -85,B 0,C 180,E1 20910.339,E2 20910.339} C_VEL
LIN {X 0,Y 577.253,Z 419.313,A -85,B 0,C 180,E1 20907.212,E2 20907.212} C_VEL
LIN {X 0,Y 577.317,Z 419.29,A -85,B 0,C 180,E1 20904.017,E2 20904.017} C_VEL
LIN {X 0,Y 577.245,Z 419.283,A -85,B 0,C 180,E1 20900.906,E2 20900.906} C_VEL
LIN {X 0,Y 577.32,Z 419.319,A -85,B 0,C 180,E1 20897.735,E2 20897.735} C_VEL
LIN {X 0,Y 577.24,Z 419.274,A -85,B 0,C 180,E1 20894.649,E2 20894.649} C_VEL
LIN {X 0,Y 577.315,Z 419.316,A -85,B 0,C 180,E1 20891.489,E2 20891.489} C_VEL
LIN {X 0,Y 577.24,Z 419.276,A -85,B 0,C 180,E1 20888.367,E2 20888.367} C_VEL
LIN {X 0,Y 577.313,Z 419.312,A -85,B 0,C 180,E1 20885.263,E2 20885.263} C_VEL
LIN {X 0,Y 577.237,Z 419.279,A -85,B 0,C 180,E1 20882.085,E2 20882.085} C_VEL
LIN {X 0,Y 577.299,Z 419.31,A -85,B 0,C 180,E1 20878.908,E2 20878.908} C_VEL
LIN {X 0,Y 577.237,Z 419.282,A -85,B 0,C 180,E1 20875.828,E2 20875.828} C_VEL
LIN {X 0,Y 577.291,Z 419.307,A -85,B 0,C 180,E1 20872.636,E2 20872.636} C_VEL
LIN {X 0,Y 577.233,Z 419.287,A -85,B 0,C 180,E1 20869.621,E2 20869.621} C_VEL
LIN {X 0,Y 577.295,Z 419.298,A -85,B 0,C 180,E1 20866.478,E2 20866.478} C_VEL
LIN {X 0,Y 577.231,Z 419.297,A -85,B 0,C 180,E1 20863.496,E2 20863.496} C_VEL
LIN {X 0,Y 577.301,Z 419.275,A -85,B 0,C 180,E1 20860.366,E2 20860.366} C_VEL
LIN {X 0,Y 577.232,Z 419.324,A -85,B 0,C 180,E1 20857.276,E2 20857.276} C_VEL
LIN {X 0,Y 577.296,Z 419.275,A -85,B 0,C 180,E1 20854.121,E2 20854.121} C_VEL
LIN {X 0,Y 577.226,Z 419.301,A -85,B 0,C 180,E1 20851.099,E2 20851.099} C_VEL
LIN {X 0,Y 577.287,Z 419.424,A -85,B 0,C 180,E1 20850.388,E2 20850.388} C_VEL
LIN {X 0,Y 578.704,Z 422.963,A -85,B 0,C 180,E1 20849.7,E2 20849.7} C_VEL
LIN {X 0,Y 579.869,Z 424.562,A -85,B 0,C 180,E1 20849.309,E2 20849.309} C_VEL
LIN {X 0,Y 580.81,Z 426.72,A -85,B 0,C 180,E1 20848.962,E2 20848.962} C_VEL
LIN {X 0,Y 584.515,Z 431.185,A -85,B 0,C 180,E1 20848.263,E2 20848.263} C_VEL
LIN {X 0,Y 592.831,Z 441.788,A -85,B 0,C 180,E1 20846.759,E2 20846.759} C_VEL
LIN {X 0,Y 603.732,Z 456.264,A -85,B 0,C 180,E1 20844.922,E2 20844.922} C_VEL
LIN {X 0,Y 615.35,Z 472.592,A -85,B 0,C 180,E1 20843.101,E2 20843.101} C_VEL
LIN {X 0,Y 624.02,Z 485.373,A -85,B 0,C 180,E1 20841.822,E2 20841.822} C_VEL
LIN {X 0,Y 629.719,Z 494.155,A -85,B 0,C 180,E1 20841.013,E2 20841.013} C_VEL
LIN {X 0,Y 623.986,Z 695.536,A -85,B 0,C 180,E1 20838.146,E2 20838.146} C_VEL
LIN {X 0,Y 618.325,Z 902.683,A -85,B 0,C 180,E1 20835.249,E2 20835.249} C_VEL
LIN {X 0,Y 617.109,Z 925.196,A -85,B 0,C 180,E1 20834.849,E2 20834.849} C_VEL
LIN {X 0,Y 615.199,Z 952.228,A -85,B 0,C 180,E1 20834.212,E2 20834.212} C_VEL
LIN {X 0,Y 612.944,Z 976.913,A -85,B 0,C 180,E1 20833.454,E2 20833.454} C_VEL
LIN {X 0,Y 610.785,Z 997.73,A -85,B 0,C 180,E1 20832.689,E2 20832.689} C_VEL
LIN {X 0,Y 608.55,Z 1017.624,A -85,B 0,C 180,E1 20831.836,E2 20831.836} C_VEL
LIN {X 0,Y 606.27,Z 1035.978,A -85,B 0,C 180,E1 20830.943,E2 20830.943} C_VEL
LIN {X 0,Y 603.653,Z 1055.594,A -85,B 0,C 180,E1 20829.862,E2 20829.862} C_VEL
LIN {X 0,Y 600.511,Z 1078.166,A -85,B 0,C 180,E1 20828.449,E2 20828.449} C_VEL
LIN {X 0,Y 597.043,Z 1101.269,A -85,B 0,C 180,E1 20826.773,E2 20826.773} C_VEL
LIN {X 0,Y 594.323,Z 1119.071,A -85,B 0,C 180,E1 20825.317,E2 20825.317} C_VEL
LIN {X 0,Y 591.69,Z 1136.264,A -85,B 0,C 180,E1 20823.754,E2 20823.754} C_VEL
LIN {X 0,Y 588.93,Z 1154.54,A -85,B 0,C 180,E1 20821.907,E2 20821.907} C_VEL
LIN {X 0,Y 586.029,Z 1174.171,A -85,B 0,C 180,E1 20819.652,E2 20819.652} C_VEL
LIN {X 0,Y 583.828,Z 1189.638,A -85,B 0,C 180,E1 20817.649,E2 20817.649} C_VEL
LIN {X 0,Y 581.912,Z 1204.206,A -85,B 0,C 180,E1 20815.545,E2 20815.545} C_VEL
LIN {X 0,Y 579.94,Z 1220.724,A -85,B 0,C 180,E1 20812.821,E2 20812.821} C_VEL
LIN {X 0,Y 578.702,Z 1232.283,A -85,B 0,C 180,E1 20810.635,E2 20810.635} C_VEL
LIN {X 0,Y 577.743,Z 1242.46,A -85,B 0,C 180,E1 20808.46,E2 20808.46} C_VEL
LIN {X 0,Y 576.967,Z 1252.975,A -85,B 0,C 180,E1 20805.882,E2 20805.882} C_VEL
LIN {X 0,Y 576.446,Z 1261.848,A -85,B 0,C 180,E1 20803.232,E2 20803.232} C_VEL
LIN {X 0,Y 576.157,Z 1268.064,A -85,B 0,C 180,E1 20801.002,E2 20801.002} C_VEL
LIN {X 0,Y 576.012,Z 1273.136,A -85,B 0,C 180,E1 20798.783,E2 20798.783} C_VEL
LIN {X 0,Y 575.945,Z 1277.639,A -85,B 0,C 180,E1 20796.176,E2 20796.176} C_VEL
LIN {X 0,Y 575.913,Z 1280.473,A -85,B 0,C 180,E1 20793.58,E2 20793.58} C_VEL
LIN {X 0,Y 575.895,Z 1281.714,A -85,B 0,C 180,E1 20791.29,E2 20791.29} C_VEL
LIN {X 0,Y 575.865,Z 1281.826,A -85,B 0,C 180,E1 20789.201,E2 20789.201} C_VEL
LIN {X 0,Y 575.91,Z 1281.013,A -85,B 0,C 180,E1 20787.211,E2 20787.211} C_VEL
LIN {X 0,Y 575.92,Z 1279.105,A -85,B 0,C 180,E1 20785.017,E2 20785.017} C_VEL
LIN {X 0,Y 575.961,Z 1275.897,A -85,B 0,C 180,E1 20782.717,E2 20782.717} C_VEL
LIN {X 0,Y 576.06,Z 1270.812,A -85,B 0,C 180,E1 20780.103,E2 20780.103} C_VEL
LIN {X 0,Y 576.326,Z 1263.951,A -85,B 0,C 180,E1 20777.473,E2 20777.473} C_VEL
LIN {X 0,Y 576.716,Z 1256.853,A -85,B 0,C 180,E1 20775.232,E2 20775.232} C_VEL
LIN {X 0,Y 577.237,Z 1248.887,A -85,B 0,C 180,E1 20773.079,E2 20773.079} C_VEL
LIN {X 0,Y 578.042,Z 1239.22,A -85,B 0,C 180,E1 20770.811,E2 20770.811} C_VEL
LIN {X 0,Y 579.36,Z 1225.855,A -85,B 0,C 180,E1 20768.111,E2 20768.111} C_VEL
LIN {X 0,Y 580.815,Z 1212.899,A -85,B 0,C 180,E1 20765.841,E2 20765.841} C_VEL
LIN {X 0,Y 582.458,Z 1199.963,A -85,B 0,C 180,E1 20763.819,E2 20763.819} C_VEL
LIN {X 0,Y 584.738,Z 1183.397,A -85,B 0,C 180,E1 20761.503,E2 20761.503} C_VEL
LIN {X 0,Y 587.334,Z 1165.201,A -85,B 0,C 180,E1 20759.286,E2 20759.286} C_VEL
LIN {X 0,Y 589.714,Z 1149.283,A -85,B 0,C 180,E1 20757.545,E2 20757.545} C_VEL
LIN {X 0,Y 592.344,Z 1132.139,A -85,B 0,C 180,E1 20755.855,E2 20755.855} C_VEL
LIN {X 0,Y 595.739,Z 1109.865,A -85,B 0,C 180,E1 20753.904,E2 20753.904} C_VEL
LIN {X 0,Y 598.81,Z 1089.191,A -85,B 0,C 180,E1 20752.325,E2 20752.325} C_VEL
LIN {X 0,Y 601.608,Z 1069.952,A -85,B 0,C 180,E1 20751.017,E2 20751.017} C_VEL
LIN {X 0,Y 604.647,Z 1048.29,A -85,B 0,C 180,E1 20749.714,E2 20749.714} C_VEL
LIN {X 0,Y 608.023,Z 1022.03,A -85,B 0,C 180,E1 20748.364,E2 20748.364} C_VEL
LIN {X 0,Y 610.461,Z 1000.724,A -85,B 0,C 180,E1 20747.431,E2 20747.431} C_VEL
LIN {X 0,Y 612.608,Z 980.186,A -85,B 0,C 180,E1 20746.658,E2 20746.658} C_VEL
LIN {X 0,Y 614.55,Z 959.138,A -85,B 0,C 180,E1 20745.987,E2 20745.987} C_VEL
LIN {X 0,Y 616.409,Z 935.866,A -85,B 0,C 180,E1 20745.381,E2 20745.381} C_VEL
LIN {X 0,Y 618.148,Z 906.899,A -85,B 0,C 180,E1 20744.815,E2 20744.815} C_VEL
LIN {X 0,Y 619.858,Z 849.638,A -85,B 0,C 180,E1 20744.002,E2 20744.002} C_VEL
LIN {X 0,Y 625.776,Z 631.087,A -85,B 0,C 180,E1 20740.944,E2 20740.944} C_VEL
LIN {X 0,Y 629.712,Z 493.825,A -85,B 0,C 180,E1 20738.981,E2 20738.981} C_VEL
LIN {X 0,Y 616.394,Z 474.1,A -85,B 0,C 180,E1 20737.059,E2 20737.059} C_VEL
LIN {X 0,Y 605.483,Z 458.724,A -85,B 0,C 180,E1 20735.367,E2 20735.367} C_VEL
LIN {X 0,Y 598.675,Z 449.628,A -85,B 0,C 180,E1 20734.253,E2 20734.253} C_VEL
LIN {X 0,Y 591.354,Z 439.807,A -85,B 0,C 180,E1 20732.988,E2 20732.988} C_VEL
LIN {X 0,Y 582.843,Z 429.129,A -85,B 0,C 180,E1 20731.435,E2 20731.435} C_VEL
LIN {X 0,Y 580.179,Z 425.57,A -85,B 0,C 180,E1 20730.877,E2 20730.877} C_VEL
LIN {X 0,Y 579.577,Z 423.988,A -85,B 0,C 180,E1 20730.584,E2 20730.584} C_VEL
LIN {X 0,Y 577.516,Z 420.453,A -85,B 0,C 180,E1 20729.795,E2 20729.795} C_VEL
LIN {X 0,Y 577.259,Z 419.282,A -85,B 0,C 180,E1 20729.581,E2 20729.581} C_VEL
